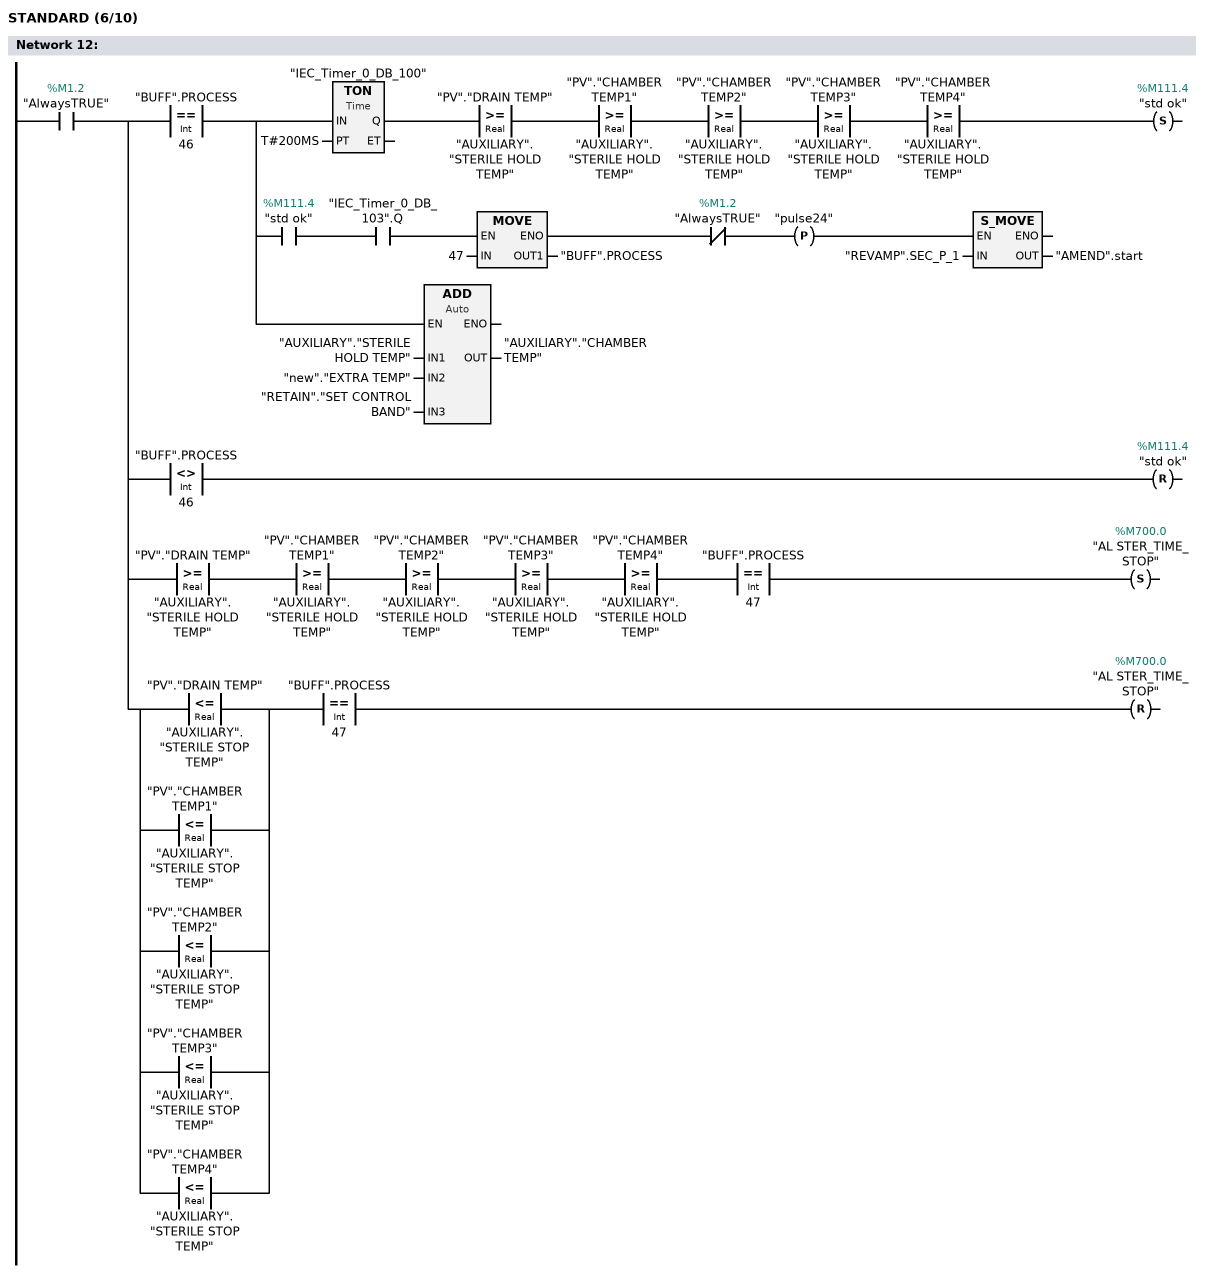
   RUNG wire#powerrail
      Contact( "AlwaysTRUE" )
      wire#w1
      { S7_Templates := "SrcType := Int" } EQ_Contact(in1 := "BUFF".PROCESS, in2 := 46)
      wire#w2
      { S7_Templates := "time_type := Time" } "IEC_Timer_0_DB_100".TON(pt := T#200MS, et =>)
      { S7_Templates := "SrcType := Real" } GE_Contact(in1 := "PV"."DRAIN TEMP", in2 := "AUXILIARY"."STERILE HOLD TEMP")
      { S7_Templates := "SrcType := Real" } GE_Contact(in1 := "PV"."CHAMBER TEMP1", in2 := "AUXILIARY"."STERILE HOLD TEMP")
      { S7_Templates := "SrcType := Real" } GE_Contact(in1 := "PV"."CHAMBER TEMP2", in2 := "AUXILIARY"."STERILE HOLD TEMP")
      { S7_Templates := "SrcType := Real" } GE_Contact(in1 := "PV"."CHAMBER TEMP3", in2 := "AUXILIARY"."STERILE HOLD TEMP")
      { S7_Templates := "SrcType := Real" } GE_Contact(in1 := "PV"."CHAMBER TEMP4", in2 := "AUXILIARY"."STERILE HOLD TEMP")
      S_Coil( "std ok" )
   END_RUNG
   RUNG wire#w2
      Contact( "std ok" )
      Contact( "IEC_Timer_0_DB_103".Q )
      Move(in := 47, out1 => "BUFF".PROCESS)
      I_Contact( "AlwaysTRUE" )
      P_Trig( "pulse24" )
      S_Move(in := "REVAMP".SEC_P_1, out => "AMEND".start)
   END_RUNG
   RUNG wire#w2
      Add(in1 := "AUXILIARY"."STERILE HOLD TEMP", in2 := "new"."EXTRA TEMP", in3 := "RETAIN"."SET CONTROL BAND", out => "AUXILIARY"."CHAMBER TEMP")
   END_RUNG
   RUNG wire#w1
      { S7_Templates := "SrcType := Int" } NE_Contact(in1 := "BUFF".PROCESS, in2 := 46)
      R_Coil( "std ok" )
   END_RUNG
   RUNG wire#w1
      { S7_Templates := "SrcType := Real" } GE_Contact(in1 := "PV"."DRAIN TEMP", in2 := "AUXILIARY"."STERILE HOLD TEMP")
      { S7_Templates := "SrcType := Real" } GE_Contact(in1 := "PV"."CHAMBER TEMP1", in2 := "AUXILIARY"."STERILE HOLD TEMP")
      { S7_Templates := "SrcType := Real" } GE_Contact(in1 := "PV"."CHAMBER TEMP2", in2 := "AUXILIARY"."STERILE HOLD TEMP")
      { S7_Templates := "SrcType := Real" } GE_Contact(in1 := "PV"."CHAMBER TEMP3", in2 := "AUXILIARY"."STERILE HOLD TEMP")
      { S7_Templates := "SrcType := Real" } GE_Contact(in1 := "PV"."CHAMBER TEMP4", in2 := "AUXILIARY"."STERILE HOLD TEMP")
      { S7_Templates := "SrcType := Int" } EQ_Contact(in1 := "BUFF".PROCESS, in2 := 47)
      S_Coil( "AL STER_TIME_STOP" )
   END_RUNG
   RUNG wire#w1
      { S7_Templates := "SrcType := Real" } LE_Contact(in1 := "PV"."DRAIN TEMP", in2 := "AUXILIARY"."STERILE STOP TEMP")
      wire#w3
      { S7_Templates := "SrcType := Int" } EQ_Contact(in1 := "BUFF".PROCESS, in2 := 47)
      R_Coil( "AL STER_TIME_STOP" )
   END_RUNG
   RUNG wire#w1
      { S7_Templates := "SrcType := Real" } LE_Contact(in1 := "PV"."CHAMBER TEMP1", in2 := "AUXILIARY"."STERILE STOP TEMP")
   END_RUNG wire#w3
   RUNG wire#w1
      { S7_Templates := "SrcType := Real" } LE_Contact(in1 := "PV"."CHAMBER TEMP2", in2 := "AUXILIARY"."STERILE STOP TEMP")
   END_RUNG wire#w3
   RUNG wire#w1
      { S7_Templates := "SrcType := Real" } LE_Contact(in1 := "PV"."CHAMBER TEMP3", in2 := "AUXILIARY"."STERILE STOP TEMP")
   END_RUNG wire#w3
   RUNG wire#w1
      { S7_Templates := "SrcType := Real" } LE_Contact(in1 := "PV"."CHAMBER TEMP4", in2 := "AUXILIARY"."STERILE STOP TEMP")
   END_RUNG wire#w3
   // the same network as SCL:
   #_w1 := "AlwaysTRUE" AND ("BUFF".PROCESS = 46);
   "IEC_Timer_0_DB_100".TON(IN := #_w1, PT := T#200MS);
   IF "IEC_Timer_0_DB_100".Q AND ("PV"."DRAIN TEMP" >= "AUXILIARY"."STERILE HOLD TEMP") AND ("PV"."CHAMBER TEMP1" >= "AUXILIARY"."STERILE HOLD TEMP") AND ("PV"."CHAMBER TEMP2" >= "AUXILIARY"."STERILE HOLD TEMP") AND ("PV"."CHAMBER TEMP3" >= "AUXILIARY"."STERILE HOLD TEMP") AND ("PV"."CHAMBER TEMP4" >= "AUXILIARY"."STERILE HOLD TEMP") THEN
       "std ok" := TRUE;
   END_IF;
   #_w2 := #_w1 AND "std ok" AND "IEC_Timer_0_DB_103".Q;
   IF #_w2 THEN "BUFF".PROCESS := 47; END_IF;
   #_w3 := #_w2 AND NOT "AlwaysTRUE";
   #_w4 := #_w3 AND NOT "pulse24";   // rising edge
   "pulse24" := #_w3;
   IF #_w4 THEN "AMEND".start := "REVAMP".SEC_P_1; END_IF;
   IF #_w1 THEN
       "AUXILIARY"."CHAMBER TEMP" := "AUXILIARY"."STERILE HOLD TEMP" + "new"."EXTRA TEMP" + "RETAIN"."SET CONTROL BAND";
   END_IF;
   IF "AlwaysTRUE" AND ("BUFF".PROCESS <> 46) THEN "std ok" := FALSE; END_IF;
   IF "AlwaysTRUE" AND ("PV"."DRAIN TEMP" >= "AUXILIARY"."STERILE HOLD TEMP") AND ("PV"."CHAMBER TEMP1" >= "AUXILIARY"."STERILE HOLD TEMP") AND ("PV"."CHAMBER TEMP2" >= "AUXILIARY"."STERILE HOLD TEMP") AND ("PV"."CHAMBER TEMP3" >= "AUXILIARY"."STERILE HOLD TEMP") AND ("PV"."CHAMBER TEMP4" >= "AUXILIARY"."STERILE HOLD TEMP") AND ("BUFF".PROCESS = 47) THEN
       "AL STER_TIME_STOP" := TRUE;
   END_IF;
   IF "AlwaysTRUE" AND (("PV"."DRAIN TEMP" <= "AUXILIARY"."STERILE STOP TEMP") OR ("PV"."CHAMBER TEMP1" <= "AUXILIARY"."STERILE STOP TEMP") OR ("PV"."CHAMBER TEMP2" <= "AUXILIARY"."STERILE STOP TEMP") OR ("PV"."CHAMBER TEMP3" <= "AUXILIARY"."STERILE STOP TEMP") OR ("PV"."CHAMBER TEMP4" <= "AUXILIARY"."STERILE STOP TEMP")) AND ("BUFF".PROCESS = 47) THEN
       "AL STER_TIME_STOP" := FALSE;
   END_IF;
END_REGION

REGION Network 13
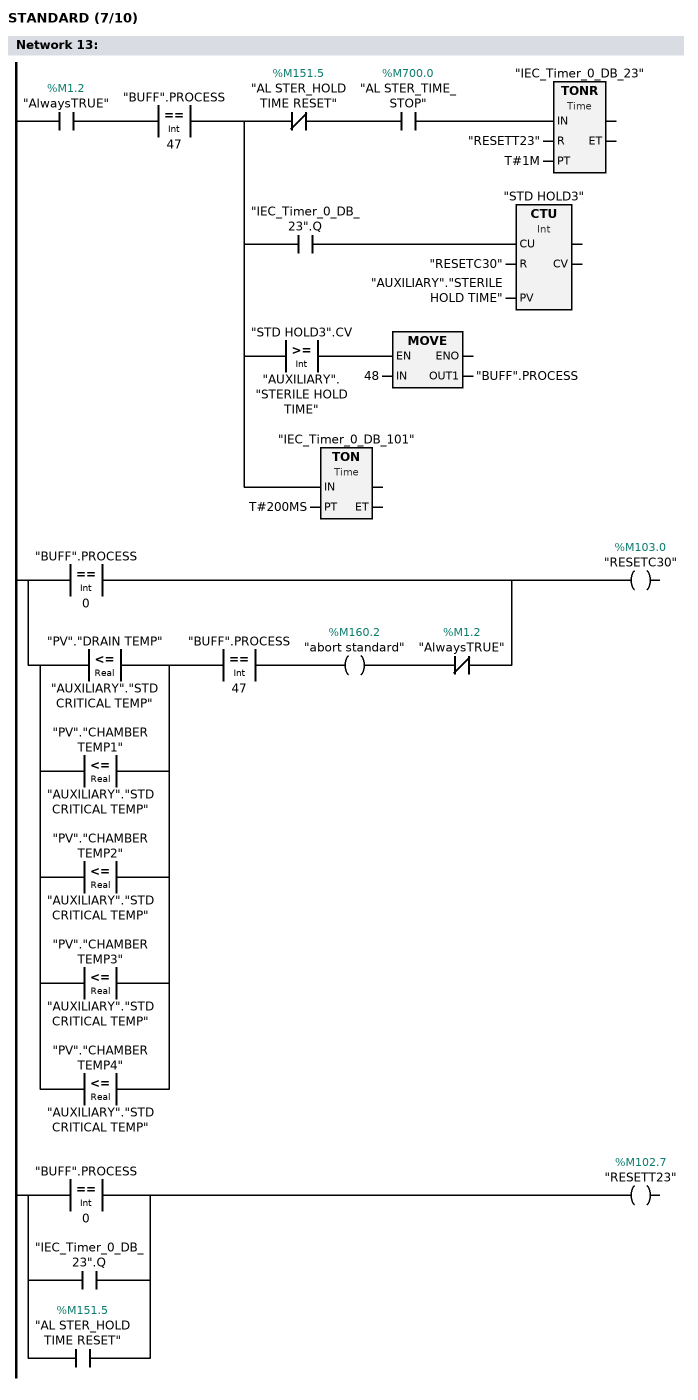
   RUNG wire#powerrail
      Contact( "AlwaysTRUE" )
      { S7_Templates := "SrcType := Int" } EQ_Contact(in1 := "BUFF".PROCESS, in2 := 47)
      wire#w1
      I_Contact( "AL STER_HOLD TIME RESET" )
      Contact( "AL STER_TIME_STOP" )
      { S7_Templates := "time_type := Time" } "IEC_Timer_0_DB_23".TONR(r := "RESETT23", pt := T#1M, et =>)
   END_RUNG
   RUNG wire#w1
      Contact( "IEC_Timer_0_DB_23".Q )
      { S7_Templates := "value_type := Int" } "STD HOLD3".CTU(r := "RESETC30", pv := "AUXILIARY"."STERILE HOLD TIME", cv =>)
   END_RUNG
   RUNG wire#w1
      { S7_Templates := "SrcType := Int" } GE_Contact(in1 := "STD HOLD3".CV, in2 := "AUXILIARY"."STERILE HOLD TIME")
      Move(in := 48, out1 => "BUFF".PROCESS)
   END_RUNG
   RUNG wire#w1
      { S7_Templates := "time_type := Time" } "IEC_Timer_0_DB_101".TON(pt := T#200MS, et =>)
   END_RUNG
   RUNG wire#powerrail
      { S7_Templates := "SrcType := Int" } EQ_Contact(in1 := "BUFF".PROCESS, in2 := 0)
      wire#w2
      Coil( "RESETC30" )
   END_RUNG
   RUNG wire#powerrail
      { S7_Templates := "SrcType := Real" } LE_Contact(in1 := "PV"."DRAIN TEMP", in2 := "AUXILIARY"."STD CRITICAL TEMP")
      wire#w3
      { S7_Templates := "SrcType := Int" } EQ_Contact(in1 := "BUFF".PROCESS, in2 := 47)
      Coil( "abort standard" )
      I_Contact( "AlwaysTRUE" )
   END_RUNG wire#w2
   RUNG wire#powerrail
      { S7_Templates := "SrcType := Real" } LE_Contact(in1 := "PV"."CHAMBER TEMP1", in2 := "AUXILIARY"."STD CRITICAL TEMP")
   END_RUNG wire#w3
   RUNG wire#powerrail
      { S7_Templates := "SrcType := Real" } LE_Contact(in1 := "PV"."CHAMBER TEMP2", in2 := "AUXILIARY"."STD CRITICAL TEMP")
   END_RUNG wire#w3
   RUNG wire#powerrail
      { S7_Templates := "SrcType := Real" } LE_Contact(in1 := "PV"."CHAMBER TEMP3", in2 := "AUXILIARY"."STD CRITICAL TEMP")
   END_RUNG wire#w3
   RUNG wire#powerrail
      { S7_Templates := "SrcType := Real" } LE_Contact(in1 := "PV"."CHAMBER TEMP4", in2 := "AUXILIARY"."STD CRITICAL TEMP")
   END_RUNG wire#w3
   RUNG wire#powerrail
      { S7_Templates := "SrcType := Int" } EQ_Contact(in1 := "BUFF".PROCESS, in2 := 0)
      wire#w4
      Coil( "RESETT23" )
   END_RUNG
   RUNG wire#powerrail
      Contact( "IEC_Timer_0_DB_23".Q )
   END_RUNG wire#w4
   RUNG wire#powerrail
      Contact( "AL STER_HOLD TIME RESET" )
   END_RUNG wire#w4
   // the same network as SCL:
   #_w1 := "AlwaysTRUE" AND ("BUFF".PROCESS = 47);
   "IEC_Timer_0_DB_23".TONR(IN := #_w1 AND NOT "AL STER_HOLD TIME RESET" AND "AL STER_TIME_STOP",
                           R := "RESETT23",
                           PT := T#1M);
   "STD HOLD3".CTU(CU := #_w1 AND "IEC_Timer_0_DB_23".Q, R := "RESETC30", PV := "AUXILIARY"."STERILE HOLD TIME");
   IF #_w1 AND ("STD HOLD3".CV >= "AUXILIARY"."STERILE HOLD TIME") THEN "BUFF".PROCESS := 48; END_IF;
   "IEC_Timer_0_DB_101".TON(IN := #_w1, PT := T#200MS);
   "abort standard" := (("PV"."DRAIN TEMP" <= "AUXILIARY"."STD CRITICAL TEMP") OR ("PV"."CHAMBER TEMP1" <= "AUXILIARY"."STD CRITICAL TEMP") OR ("PV"."CHAMBER TEMP2" <= "AUXILIARY"."STD CRITICAL TEMP") OR ("PV"."CHAMBER TEMP3" <= "AUXILIARY"."STD CRITICAL TEMP") OR ("PV"."CHAMBER TEMP4" <= "AUXILIARY"."STD CRITICAL TEMP")) AND ("BUFF".PROCESS = 47);
   "RESETC30" := ("BUFF".PROCESS = 0) OR ("abort standard" AND NOT "AlwaysTRUE");
   "RESETT23" := ("BUFF".PROCESS = 0) OR "IEC_Timer_0_DB_23".Q OR "AL STER_HOLD TIME RESET";
END_REGION

REGION Network 14
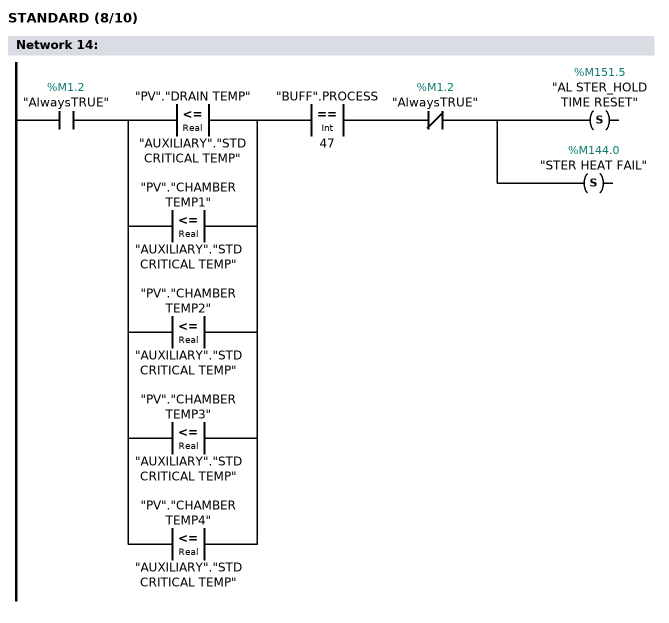
   RUNG wire#powerrail
      Contact( "AlwaysTRUE" )
      wire#w1
      { S7_Templates := "SrcType := Real" } LE_Contact(in1 := "PV"."DRAIN TEMP", in2 := "AUXILIARY"."STD CRITICAL TEMP")
      wire#w2
      { S7_Templates := "SrcType := Int" } EQ_Contact(in1 := "BUFF".PROCESS, in2 := 47)
      I_Contact( "AlwaysTRUE" )
      wire#w3
      S_Coil( "AL STER_HOLD TIME RESET" )
   END_RUNG
   RUNG wire#w1
      { S7_Templates := "SrcType := Real" } LE_Contact(in1 := "PV"."CHAMBER TEMP1", in2 := "AUXILIARY"."STD CRITICAL TEMP")
   END_RUNG wire#w2
   RUNG wire#w1
      { S7_Templates := "SrcType := Real" } LE_Contact(in1 := "PV"."CHAMBER TEMP2", in2 := "AUXILIARY"."STD CRITICAL TEMP")
   END_RUNG wire#w2
   RUNG wire#w1
      { S7_Templates := "SrcType := Real" } LE_Contact(in1 := "PV"."CHAMBER TEMP3", in2 := "AUXILIARY"."STD CRITICAL TEMP")
   END_RUNG wire#w2
   RUNG wire#w1
      { S7_Templates := "SrcType := Real" } LE_Contact(in1 := "PV"."CHAMBER TEMP4", in2 := "AUXILIARY"."STD CRITICAL TEMP")
   END_RUNG wire#w2
   RUNG wire#w3
      S_Coil( "STER HEAT FAIL" )
   END_RUNG
   // the same network as SCL:
   IF "AlwaysTRUE" AND (("PV"."DRAIN TEMP" <= "AUXILIARY"."STD CRITICAL TEMP") OR ("PV"."CHAMBER TEMP1" <= "AUXILIARY"."STD CRITICAL TEMP") OR ("PV"."CHAMBER TEMP2" <= "AUXILIARY"."STD CRITICAL TEMP") OR ("PV"."CHAMBER TEMP3" <= "AUXILIARY"."STD CRITICAL TEMP") OR ("PV"."CHAMBER TEMP4" <= "AUXILIARY"."STD CRITICAL TEMP")) AND ("BUFF".PROCESS = 47) AND NOT "AlwaysTRUE" THEN
       "AL STER_HOLD TIME RESET" := TRUE;
       "STER HEAT FAIL" := TRUE;
   END_IF;
END_REGION

REGION Network 15
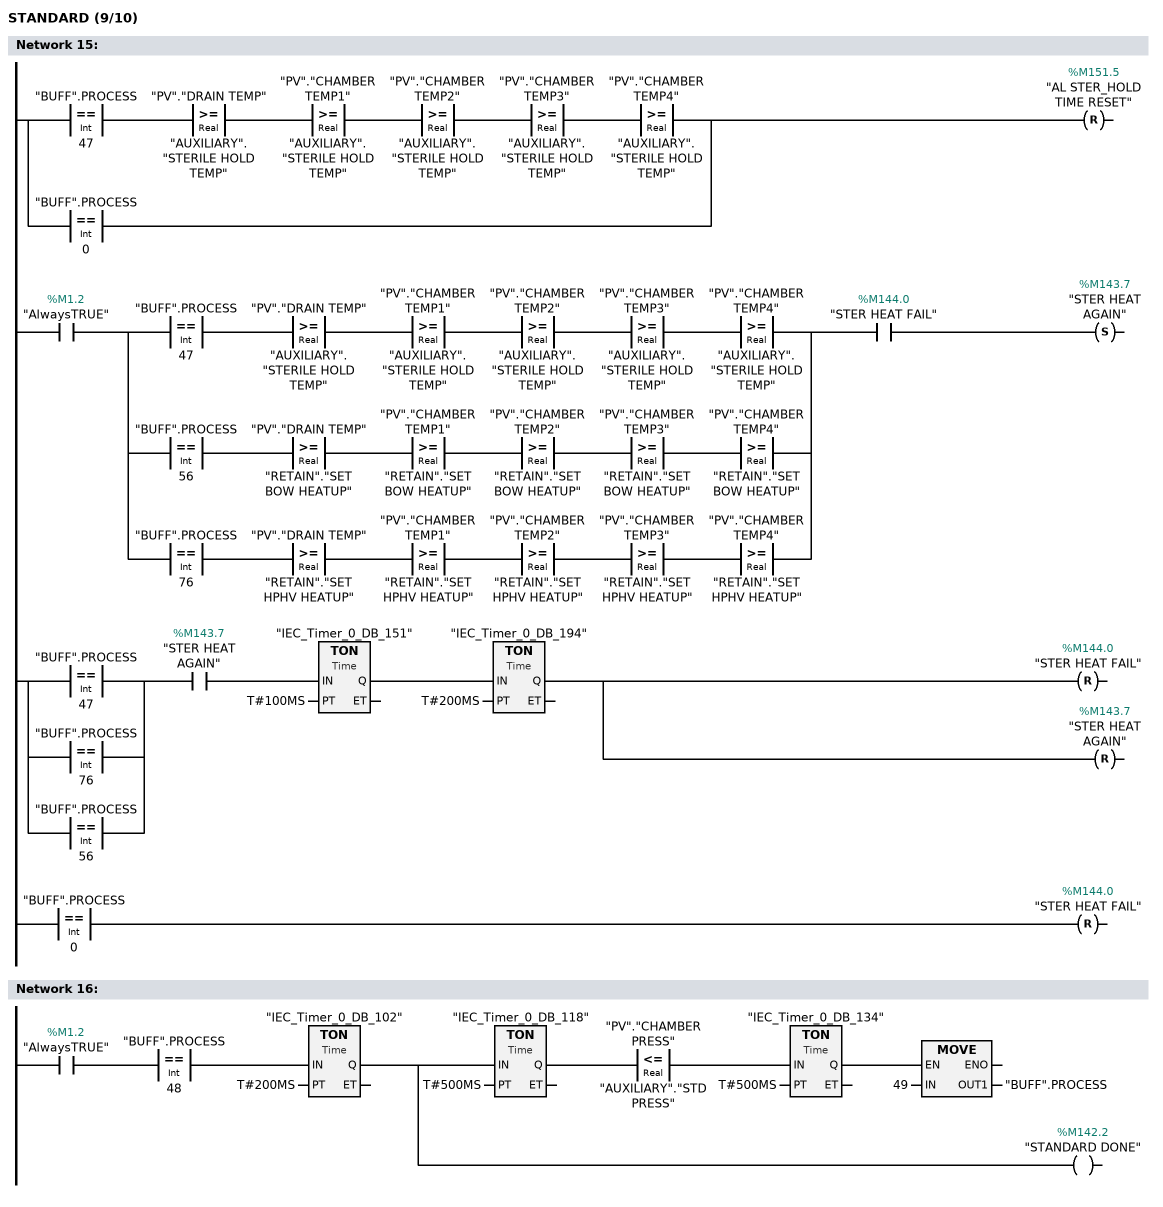
   RUNG wire#powerrail
      { S7_Templates := "SrcType := Int" } EQ_Contact(in1 := "BUFF".PROCESS, in2 := 47)
      { S7_Templates := "SrcType := Real" } GE_Contact(in1 := "PV"."DRAIN TEMP", in2 := "AUXILIARY"."STERILE HOLD TEMP")
      { S7_Templates := "SrcType := Real" } GE_Contact(in1 := "PV"."CHAMBER TEMP1", in2 := "AUXILIARY"."STERILE HOLD TEMP")
      { S7_Templates := "SrcType := Real" } GE_Contact(in1 := "PV"."CHAMBER TEMP2", in2 := "AUXILIARY"."STERILE HOLD TEMP")
      { S7_Templates := "SrcType := Real" } GE_Contact(in1 := "PV"."CHAMBER TEMP3", in2 := "AUXILIARY"."STERILE HOLD TEMP")
      { S7_Templates := "SrcType := Real" } GE_Contact(in1 := "PV"."CHAMBER TEMP4", in2 := "AUXILIARY"."STERILE HOLD TEMP")
      wire#w1
      R_Coil( "AL STER_HOLD TIME RESET" )
   END_RUNG
   RUNG wire#powerrail
      { S7_Templates := "SrcType := Int" } EQ_Contact(in1 := "BUFF".PROCESS, in2 := 0)
   END_RUNG wire#w1
   RUNG wire#powerrail
      Contact( "AlwaysTRUE" )
      wire#w2
      { S7_Templates := "SrcType := Int" } EQ_Contact(in1 := "BUFF".PROCESS, in2 := 47)
      { S7_Templates := "SrcType := Real" } GE_Contact(in1 := "PV"."DRAIN TEMP", in2 := "AUXILIARY"."STERILE HOLD TEMP")
      { S7_Templates := "SrcType := Real" } GE_Contact(in1 := "PV"."CHAMBER TEMP1", in2 := "AUXILIARY"."STERILE HOLD TEMP")
      { S7_Templates := "SrcType := Real" } GE_Contact(in1 := "PV"."CHAMBER TEMP2", in2 := "AUXILIARY"."STERILE HOLD TEMP")
      { S7_Templates := "SrcType := Real" } GE_Contact(in1 := "PV"."CHAMBER TEMP3", in2 := "AUXILIARY"."STERILE HOLD TEMP")
      { S7_Templates := "SrcType := Real" } GE_Contact(in1 := "PV"."CHAMBER TEMP4", in2 := "AUXILIARY"."STERILE HOLD TEMP")
      wire#w3
      Contact( "STER HEAT FAIL" )
      S_Coil( "STER HEAT AGAIN" )
   END_RUNG
   RUNG wire#w2
      { S7_Templates := "SrcType := Int" } EQ_Contact(in1 := "BUFF".PROCESS, in2 := 56)
      { S7_Templates := "SrcType := Real" } GE_Contact(in1 := "PV"."DRAIN TEMP", in2 := "RETAIN"."SET BOW HEATUP")
      { S7_Templates := "SrcType := Real" } GE_Contact(in1 := "PV"."CHAMBER TEMP1", in2 := "RETAIN"."SET BOW HEATUP")
      { S7_Templates := "SrcType := Real" } GE_Contact(in1 := "PV"."CHAMBER TEMP2", in2 := "RETAIN"."SET BOW HEATUP")
      { S7_Templates := "SrcType := Real" } GE_Contact(in1 := "PV"."CHAMBER TEMP3", in2 := "RETAIN"."SET BOW HEATUP")
      { S7_Templates := "SrcType := Real" } GE_Contact(in1 := "PV"."CHAMBER TEMP4", in2 := "RETAIN"."SET BOW HEATUP")
   END_RUNG wire#w3
   RUNG wire#w2
      { S7_Templates := "SrcType := Int" } EQ_Contact(in1 := "BUFF".PROCESS, in2 := 76)
      { S7_Templates := "SrcType := Real" } GE_Contact(in1 := "PV"."DRAIN TEMP", in2 := "RETAIN"."SET HPHV HEATUP")
      { S7_Templates := "SrcType := Real" } GE_Contact(in1 := "PV"."CHAMBER TEMP1", in2 := "RETAIN"."SET HPHV HEATUP")
      { S7_Templates := "SrcType := Real" } GE_Contact(in1 := "PV"."CHAMBER TEMP2", in2 := "RETAIN"."SET HPHV HEATUP")
      { S7_Templates := "SrcType := Real" } GE_Contact(in1 := "PV"."CHAMBER TEMP3", in2 := "RETAIN"."SET HPHV HEATUP")
      { S7_Templates := "SrcType := Real" } GE_Contact(in1 := "PV"."CHAMBER TEMP4", in2 := "RETAIN"."SET HPHV HEATUP")
   END_RUNG wire#w3
   RUNG wire#powerrail
      { S7_Templates := "SrcType := Int" } EQ_Contact(in1 := "BUFF".PROCESS, in2 := 47)
      wire#w4
      Contact( "STER HEAT AGAIN" )
      { S7_Templates := "time_type := Time" } "IEC_Timer_0_DB_151".TON(pt := T#100MS, et =>)
      { S7_Templates := "time_type := Time" } "IEC_Timer_0_DB_194".TON(pt := T#200MS, et =>)
      wire#w5
      R_Coil( "STER HEAT FAIL" )
   END_RUNG
   RUNG wire#powerrail
      { S7_Templates := "SrcType := Int" } EQ_Contact(in1 := "BUFF".PROCESS, in2 := 76)
   END_RUNG wire#w4
   RUNG wire#powerrail
      { S7_Templates := "SrcType := Int" } EQ_Contact(in1 := "BUFF".PROCESS, in2 := 56)
   END_RUNG wire#w4
   RUNG wire#w5
      R_Coil( "STER HEAT AGAIN" )
   END_RUNG
   RUNG wire#powerrail
      { S7_Templates := "SrcType := Int" } EQ_Contact(in1 := "BUFF".PROCESS, in2 := 0)
      R_Coil( "STER HEAT FAIL" )
   END_RUNG
   // the same network as SCL:
   IF (("BUFF".PROCESS = 47) AND ("PV"."DRAIN TEMP" >= "AUXILIARY"."STERILE HOLD TEMP") AND ("PV"."CHAMBER TEMP1" >= "AUXILIARY"."STERILE HOLD TEMP") AND ("PV"."CHAMBER TEMP2" >= "AUXILIARY"."STERILE HOLD TEMP") AND ("PV"."CHAMBER TEMP3" >= "AUXILIARY"."STERILE HOLD TEMP") AND ("PV"."CHAMBER TEMP4" >= "AUXILIARY"."STERILE HOLD TEMP")) OR ("BUFF".PROCESS = 0) THEN
       "AL STER_HOLD TIME RESET" := FALSE;
   END_IF;
   IF "AlwaysTRUE" AND ((("BUFF".PROCESS = 47) AND ("PV"."DRAIN TEMP" >= "AUXILIARY"."STERILE HOLD TEMP") AND ("PV"."CHAMBER TEMP1" >= "AUXILIARY"."STERILE HOLD TEMP") AND ("PV"."CHAMBER TEMP2" >= "AUXILIARY"."STERILE HOLD TEMP") AND ("PV"."CHAMBER TEMP3" >= "AUXILIARY"."STERILE HOLD TEMP") AND ("PV"."CHAMBER TEMP4" >= "AUXILIARY"."STERILE HOLD TEMP")) OR (("BUFF".PROCESS = 56) AND ("PV"."DRAIN TEMP" >= "RETAIN"."SET BOW HEATUP") AND ("PV"."CHAMBER TEMP1" >= "RETAIN"."SET BOW HEATUP") AND ("PV"."CHAMBER TEMP2" >= "RETAIN"."SET BOW HEATUP") AND ("PV"."CHAMBER TEMP3" >= "RETAIN"."SET BOW HEATUP") AND ("PV"."CHAMBER TEMP4" >= "RETAIN"."SET BOW HEATUP")) OR (("BUFF".PROCESS = 76) AND ("PV"."DRAIN TEMP" >= "RETAIN"."SET HPHV HEATUP") AND ("PV"."CHAMBER TEMP1" >= "RETAIN"."SET HPHV HEATUP") AND ("PV"."CHAMBER TEMP2" >= "RETAIN"."SET HPHV HEATUP") AND ("PV"."CHAMBER TEMP3" >= "RETAIN"."SET HPHV HEATUP") AND ("PV"."CHAMBER TEMP4" >= "RETAIN"."SET HPHV HEATUP"))) AND "STER HEAT FAIL" THEN
       "STER HEAT AGAIN" := TRUE;
   END_IF;
   "IEC_Timer_0_DB_151".TON(IN := (("BUFF".PROCESS = 47) OR ("BUFF".PROCESS = 76) OR ("BUFF".PROCESS = 56)) AND "STER HEAT AGAIN",
                           PT := T#100MS);
   "IEC_Timer_0_DB_194".TON(IN := "IEC_Timer_0_DB_151".Q, PT := T#200MS);
   IF "IEC_Timer_0_DB_194".Q THEN
       "STER HEAT FAIL" := FALSE;
       "STER HEAT AGAIN" := FALSE;
   END_IF;
   IF "BUFF".PROCESS = 0 THEN "STER HEAT FAIL" := FALSE; END_IF;
END_REGION

REGION Network 16
   RUNG wire#powerrail
      Contact( "AlwaysTRUE" )
      { S7_Templates := "SrcType := Int" } EQ_Contact(in1 := "BUFF".PROCESS, in2 := 48)
      { S7_Templates := "time_type := Time" } "IEC_Timer_0_DB_102".TON(pt := T#200MS, et =>)
      wire#w1
      { S7_Templates := "time_type := Time" } "IEC_Timer_0_DB_118".TON(pt := T#500MS, et =>)
      { S7_Templates := "SrcType := Real" } LE_Contact(in1 := "PV"."CHAMBER PRESS", in2 := "AUXILIARY"."STD PRESS")
      { S7_Templates := "time_type := Time" } "IEC_Timer_0_DB_134".TON(pt := T#500MS, et =>)
      Move(in := 49, out1 => "BUFF".PROCESS)
   END_RUNG
   RUNG wire#w1
      Coil( "STANDARD DONE" )
   END_RUNG
   // the same network as SCL:
   "IEC_Timer_0_DB_102".TON(IN := "AlwaysTRUE" AND ("BUFF".PROCESS = 48), PT := T#200MS);
   "IEC_Timer_0_DB_118".TON(IN := "IEC_Timer_0_DB_102".Q, PT := T#500MS);
   "IEC_Timer_0_DB_134".TON(IN := "IEC_Timer_0_DB_118".Q AND ("PV"."CHAMBER PRESS" <= "AUXILIARY"."STD PRESS"),
                           PT := T#500MS);
   IF "IEC_Timer_0_DB_134".Q THEN "BUFF".PROCESS := 49; END_IF;
   "STANDARD DONE" := "IEC_Timer_0_DB_102".Q;
END_REGION

REGION Network 17
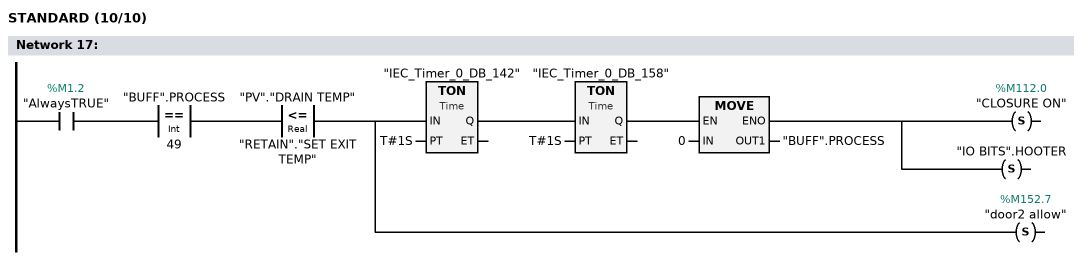
   RUNG wire#powerrail
      Contact( "AlwaysTRUE" )
      { S7_Templates := "SrcType := Int" } EQ_Contact(in1 := "BUFF".PROCESS, in2 := 49)
      { S7_Templates := "SrcType := Real" } LE_Contact(in1 := "PV"."DRAIN TEMP", in2 := "RETAIN"."SET EXIT TEMP")
      wire#w1
      { S7_Templates := "time_type := Time" } "IEC_Timer_0_DB_142".TON(pt := T#1S, et =>)
      { S7_Templates := "time_type := Time" } "IEC_Timer_0_DB_158".TON(pt := T#1S, et =>)
      Move(in := 0, out1 => "BUFF".PROCESS)
      wire#w2
      S_Coil( "CLOSURE ON" )
   END_RUNG
   RUNG wire#w2
      S_Coil( "IO BITS".HOOTER )
   END_RUNG
   RUNG wire#w1
      S_Coil( "door2 allow" )
   END_RUNG
   // the same network as SCL:
   #_w1 := "AlwaysTRUE" AND ("BUFF".PROCESS = 49) AND ("PV"."DRAIN TEMP" <= "RETAIN"."SET EXIT TEMP");
   "IEC_Timer_0_DB_142".TON(IN := #_w1, PT := T#1S);
   "IEC_Timer_0_DB_158".TON(IN := "IEC_Timer_0_DB_142".Q, PT := T#1S);
   IF "IEC_Timer_0_DB_158".Q THEN
       "BUFF".PROCESS := 0;
       "CLOSURE ON" := TRUE;
       "IO BITS".HOOTER := TRUE;
   END_IF;
   IF #_w1 THEN "door2 allow" := TRUE; END_IF;
END_REGION
END_FUNCTION

FUNCTION "VACCUM" : Void   // FC12, LAD
{ S7_Optimized_Access := 'TRUE' }
// stored: SetENOAutomatically false
   VAR_TEMP
      "VACCUM DIFF" : Real;
      "VACCUM LEAK DIFF" : Real;
   END_VAR
   VAR_TEMP   // added for the SCL form of the ladder/FBD networks
      _w1 : Bool;
      _w2 : Bool;
      _w3 : Bool;
      _w4 : Bool;
      _w5 : Bool;
      _w6 : Bool;
      _w7 : Bool;
      _w8 : Bool;
      _w9 : Bool;
      _w10 : Bool;
      _w11 : Bool;
      _w12 : Bool;
      _w13 : Bool;
      _w14 : Bool;
      _w15 : Bool;
      _w16 : Bool;
      _w17 : Bool;
      _w18 : Bool;
      _w19 : Bool;
      _w20 : Bool;
   END_VAR
BEGIN

REGION Network 1
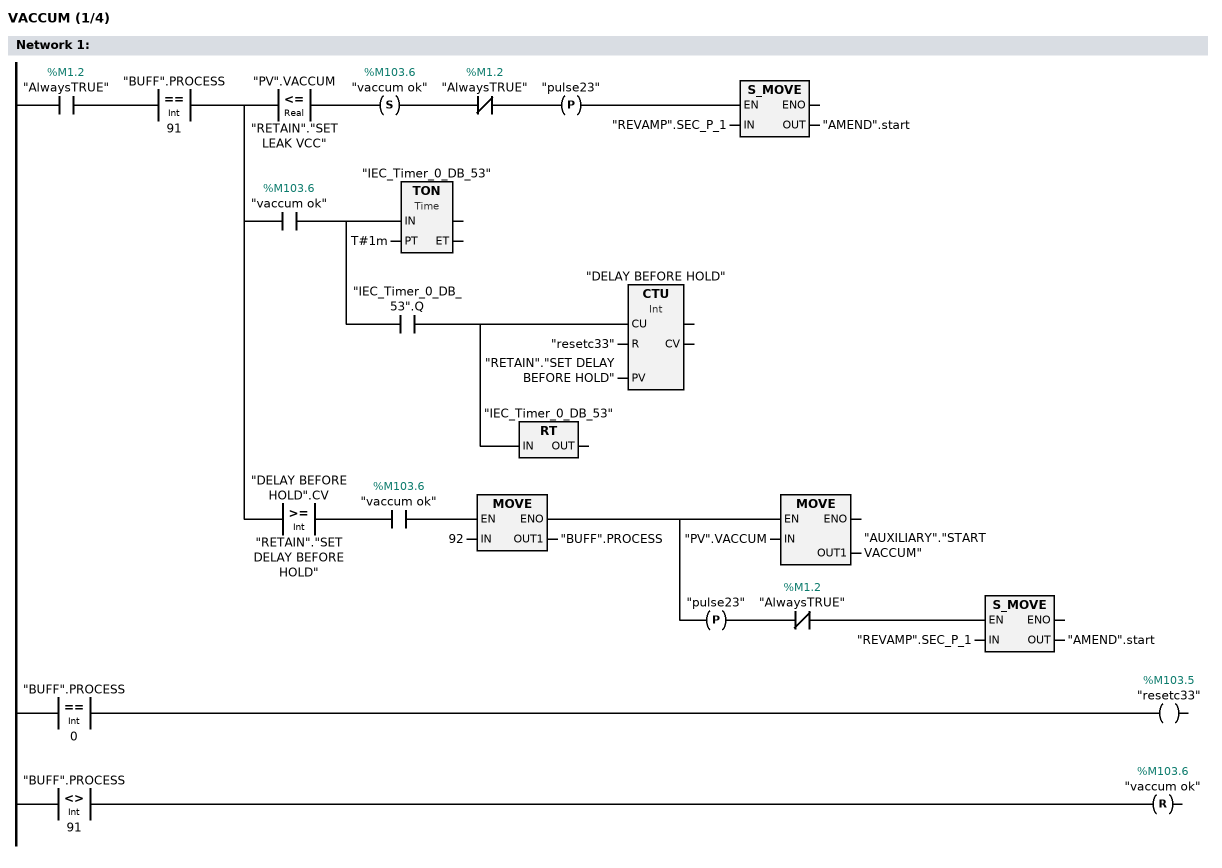
   RUNG wire#powerrail
      Contact( "AlwaysTRUE" )
      { S7_Templates := "SrcType := Int" } EQ_Contact(in1 := "BUFF".PROCESS, in2 := 91)
      wire#w1
      { S7_Templates := "SrcType := Real" } LE_Contact(in1 := "PV".VACCUM, in2 := "RETAIN"."SET LEAK VCC")
      S_Coil( "vaccum ok" )
      I_Contact( "AlwaysTRUE" )
      P_Trig( "pulse23" )
      S_Move(in := "REVAMP".SEC_P_1, out => "AMEND".start)
   END_RUNG
   RUNG wire#w1
      Contact( "vaccum ok" )
      wire#w2
      { S7_Templates := "time_type := Time" } "IEC_Timer_0_DB_53".TON(pt := T#1m, et =>)
   END_RUNG
   RUNG wire#w2
      Contact( "IEC_Timer_0_DB_53".Q )
      wire#w3
      { S7_Templates := "value_type := Int" } "DELAY BEFORE HOLD".CTU(r := "resetc33", pv := "RETAIN"."SET DELAY BEFORE HOLD", cv =>)
   END_RUNG
   RUNG wire#w3
      RT_Coil( "IEC_Timer_0_DB_53" )
   END_RUNG
   RUNG wire#w1
      { S7_Templates := "SrcType := Int" } GE_Contact(in1 := "DELAY BEFORE HOLD".CV, in2 := "RETAIN"."SET DELAY BEFORE HOLD")
      Contact( "vaccum ok" )
      Move(in := 92, out1 => "BUFF".PROCESS)
      wire#w4
      Move(in := "PV".VACCUM, out1 => "AUXILIARY"."START VACCUM")
   END_RUNG
   RUNG wire#w4
      P_Trig( "pulse23" )
      I_Contact( "AlwaysTRUE" )
      S_Move(in := "REVAMP".SEC_P_1, out => "AMEND".start)
   END_RUNG
   RUNG wire#powerrail
      { S7_Templates := "SrcType := Int" } EQ_Contact(in1 := "BUFF".PROCESS, in2 := 0)
      Coil( "resetc33" )
   END_RUNG
   RUNG wire#powerrail
      { S7_Templates := "SrcType := Int" } NE_Contact(in1 := "BUFF".PROCESS, in2 := 91)
      R_Coil( "vaccum ok" )
   END_RUNG
   // the same network as SCL:
   #_w1 := "AlwaysTRUE" AND ("BUFF".PROCESS = 91);
   #_w2 := #_w1 AND ("PV".VACCUM <= "RETAIN"."SET LEAK VCC");
   IF #_w2 THEN "vaccum ok" := TRUE; END_IF;
   #_w3 := #_w2 AND NOT "AlwaysTRUE";
   #_w4 := #_w3 AND NOT "pulse23";   // rising edge
   "pulse23" := #_w3;
   IF #_w4 THEN "AMEND".start := "REVAMP".SEC_P_1; END_IF;
   #_w5 := #_w1 AND "vaccum ok";
   "IEC_Timer_0_DB_53".TON(IN := #_w5, PT := T#1m);
   #_w6 := #_w5 AND "IEC_Timer_0_DB_53".Q;
   "DELAY BEFORE HOLD".CTU(CU := #_w6, R := "resetc33", PV := "RETAIN"."SET DELAY BEFORE HOLD");
   IF #_w6 THEN RESET_TIMER("IEC_Timer_0_DB_53"); END_IF;
   #_w7 := #_w1 AND ("DELAY BEFORE HOLD".CV >= "RETAIN"."SET DELAY BEFORE HOLD") AND "vaccum ok";
   IF #_w7 THEN
       "BUFF".PROCESS := 92;
       "AUXILIARY"."START VACCUM" := "PV".VACCUM;
   END_IF;
   #_w8 := #_w7 AND NOT "pulse23";   // rising edge
   "pulse23" := #_w7;
   IF #_w8 AND NOT "AlwaysTRUE" THEN "AMEND".start := "REVAMP".SEC_P_1; END_IF;
   "resetc33" := "BUFF".PROCESS = 0;
   IF "BUFF".PROCESS <> 91 THEN "vaccum ok" := FALSE; END_IF;
END_REGION

REGION Network 2
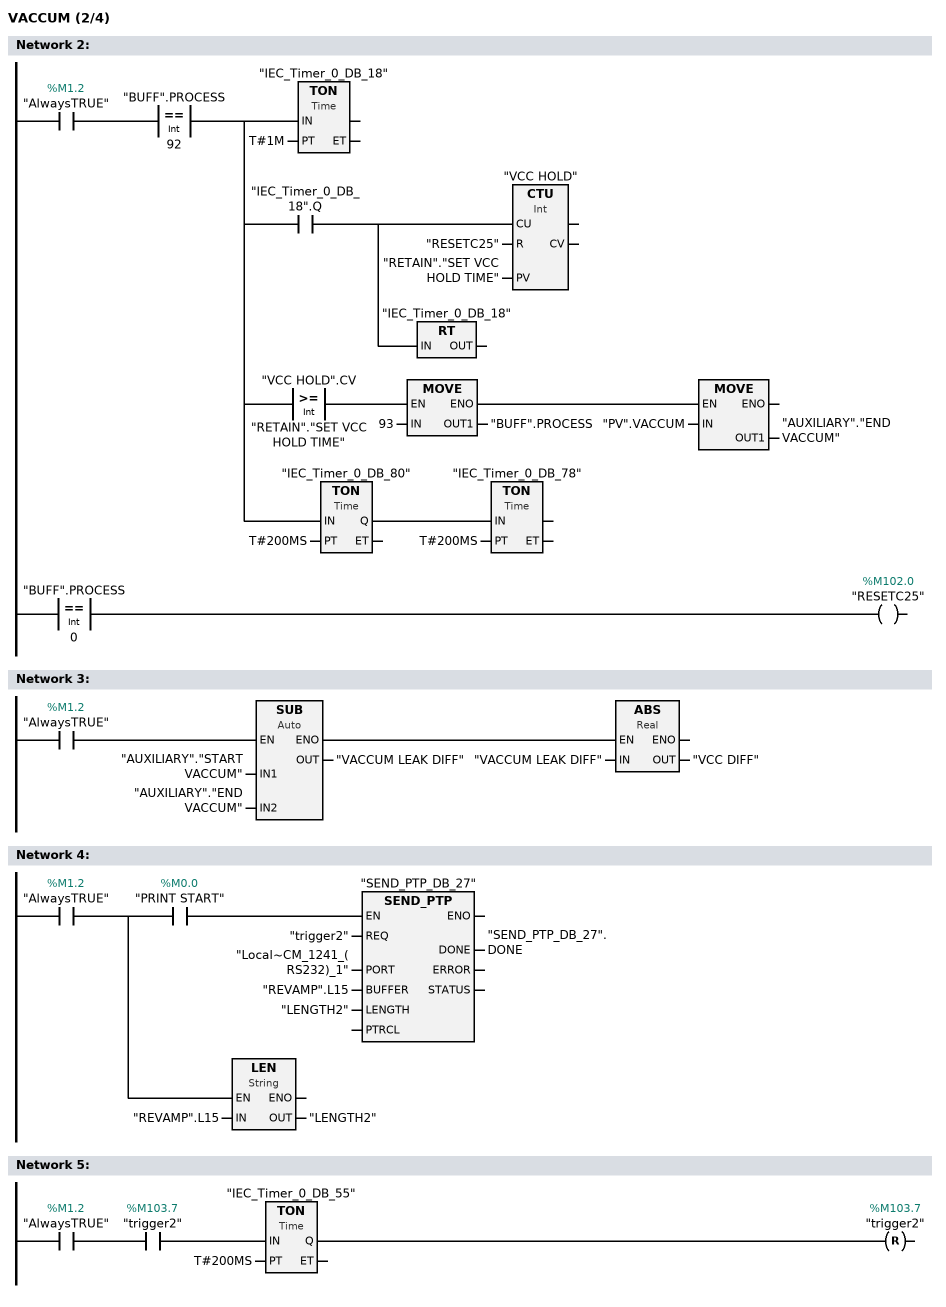
   RUNG wire#powerrail
      Contact( "AlwaysTRUE" )
      { S7_Templates := "SrcType := Int" } EQ_Contact(in1 := "BUFF".PROCESS, in2 := 92)
      wire#w1
      { S7_Templates := "time_type := Time" } "IEC_Timer_0_DB_18".TON(pt := T#1M, et =>)
   END_RUNG
   RUNG wire#w1
      Contact( "IEC_Timer_0_DB_18".Q )
      wire#w2
      { S7_Templates := "value_type := Int" } "VCC HOLD".CTU(r := "RESETC25", pv := "RETAIN"."SET VCC HOLD TIME", cv =>)
   END_RUNG
   RUNG wire#w2
      RT_Coil( "IEC_Timer_0_DB_18" )
   END_RUNG
   RUNG wire#w1
      { S7_Templates := "SrcType := Int" } GE_Contact(in1 := "VCC HOLD".CV, in2 := "RETAIN"."SET VCC HOLD TIME")
      Move(in := 93, out1 => "BUFF".PROCESS)
      Move(in := "PV".VACCUM, out1 => "AUXILIARY"."END VACCUM")
   END_RUNG
   RUNG wire#w1
      { S7_Templates := "time_type := Time" } "IEC_Timer_0_DB_80".TON(pt := T#200MS, et =>)
      { S7_Templates := "time_type := Time" } "IEC_Timer_0_DB_78".TON(pt := T#200MS, et =>)
   END_RUNG
   RUNG wire#powerrail
      { S7_Templates := "SrcType := Int" } EQ_Contact(in1 := "BUFF".PROCESS, in2 := 0)
      Coil( "RESETC25" )
   END_RUNG
   // the same network as SCL:
   #_w1 := "AlwaysTRUE" AND ("BUFF".PROCESS = 92);
   "IEC_Timer_0_DB_18".TON(IN := #_w1, PT := T#1M);
   #_w2 := #_w1 AND "IEC_Timer_0_DB_18".Q;
   "VCC HOLD".CTU(CU := #_w2, R := "RESETC25", PV := "RETAIN"."SET VCC HOLD TIME");
   IF #_w2 THEN RESET_TIMER("IEC_Timer_0_DB_18"); END_IF;
   IF #_w1 AND ("VCC HOLD".CV >= "RETAIN"."SET VCC HOLD TIME") THEN
       "BUFF".PROCESS := 93;
       "AUXILIARY"."END VACCUM" := "PV".VACCUM;
   END_IF;
   "IEC_Timer_0_DB_80".TON(IN := #_w1, PT := T#200MS);
   "IEC_Timer_0_DB_78".TON(IN := "IEC_Timer_0_DB_80".Q, PT := T#200MS);
   "RESETC25" := "BUFF".PROCESS = 0;
END_REGION

REGION Network 3
   RUNG wire#powerrail
      Contact( "AlwaysTRUE" )
      Sub(in1 := "AUXILIARY"."START VACCUM", in2 := "AUXILIARY"."END VACCUM", out => "VACCUM LEAK DIFF")
      { S7_Templates := "SrcType := Real" } Abs(in := "VACCUM LEAK DIFF", out => "VCC DIFF")
   END_RUNG
   // the same network as SCL:
   IF "AlwaysTRUE" THEN
       "VACCUM LEAK DIFF" := "AUXILIARY"."START VACCUM" - "AUXILIARY"."END VACCUM";
       "VCC DIFF" := ABS("VACCUM LEAK DIFF");
   END_IF;
END_REGION

REGION Network 4
   RUNG wire#powerrail
      Contact( "AlwaysTRUE" )
      wire#w1
      Contact( "PRINT START" )
      "SEND_PTP_DB_27".SEND_PTP(REQ := "trigger2", PORT := "Local~CM_1241_(RS232)_1", BUFFER := "REVAMP".L15, LENGTH := "LENGTH2", PTRCL :=, DONE => "SEND_PTP_DB_27".DONE, ERROR =>, STATUS =>)
   END_RUNG
   RUNG wire#w1
      { S7_Templates := "[str_type := String, return_type := Int]" } LEN(IN := "REVAMP".L15, OUT => "LENGTH2")
   END_RUNG
   // the same network as SCL:
   #_w1 := "AlwaysTRUE";
   IF "AlwaysTRUE" AND "PRINT START" THEN
       "SEND_PTP_DB_27"(REQ := "trigger2",   // SEND_PTP
                        PORT := "Local~CM_1241_(RS232)_1",
                        BUFFER := "REVAMP".L15,
                        LENGTH := "LENGTH2",
                        DONE => "SEND_PTP_DB_27".DONE);
   END_IF;
   IF #_w1 THEN LEN(IN := "REVAMP".L15, OUT => "LENGTH2"); END_IF;
END_REGION

REGION Network 5
   RUNG wire#powerrail
      Contact( "AlwaysTRUE" )
      Contact( "trigger2" )
      { S7_Templates := "time_type := Time" } "IEC_Timer_0_DB_55".TON(pt := T#200MS, et =>)
      R_Coil( "trigger2" )
   END_RUNG
   // the same network as SCL:
   "IEC_Timer_0_DB_55".TON(IN := "AlwaysTRUE" AND "trigger2", PT := T#200MS);
   IF "IEC_Timer_0_DB_55".Q THEN "trigger2" := FALSE; END_IF;
END_REGION

REGION Network 6
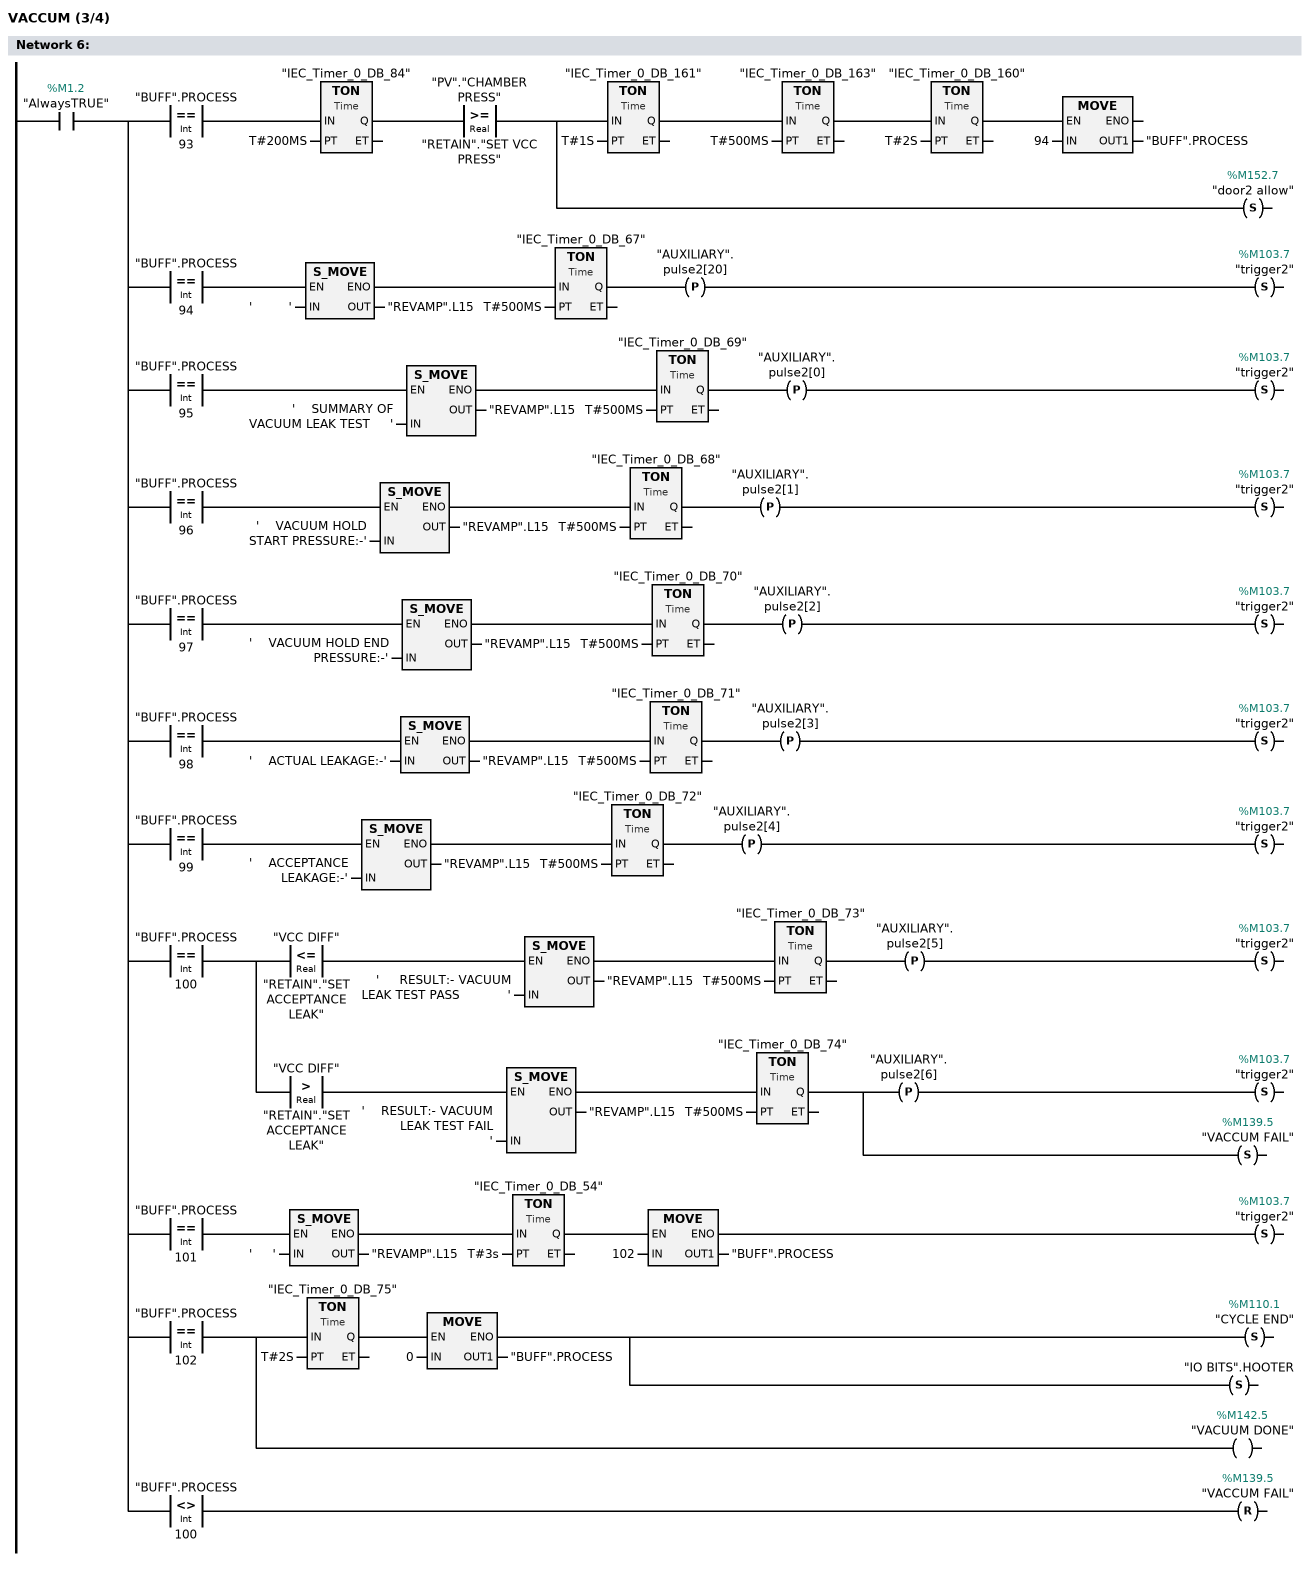
   RUNG wire#powerrail
      Contact( "AlwaysTRUE" )
      wire#w1
      { S7_Templates := "SrcType := Int" } EQ_Contact(in1 := "BUFF".PROCESS, in2 := 93)
      { S7_Templates := "time_type := Time" } "IEC_Timer_0_DB_84".TON(pt := T#200MS, et =>)
      { S7_Templates := "SrcType := Real" } GE_Contact(in1 := "PV"."CHAMBER PRESS", in2 := "RETAIN"."SET VCC PRESS")
      wire#w2
      { S7_Templates := "time_type := Time" } "IEC_Timer_0_DB_161".TON(pt := T#1S, et =>)
      { S7_Templates := "time_type := Time" } "IEC_Timer_0_DB_163".TON(pt := T#500MS, et =>)
      { S7_Templates := "time_type := Time" } "IEC_Timer_0_DB_160".TON(pt := T#2S, et =>)
      Move(in := 94, out1 => "BUFF".PROCESS)
   END_RUNG
   RUNG wire#w2
      S_Coil( "door2 allow" )
   END_RUNG
   RUNG wire#w1
      { S7_Templates := "SrcType := Int" } EQ_Contact(in1 := "BUFF".PROCESS, in2 := 94)
      S_Move(in := '         ', out => "REVAMP".L15)
      { S7_Templates := "time_type := Time" } "IEC_Timer_0_DB_67".TON(pt := T#500MS, et =>)
      P_Trig( "AUXILIARY".pulse2[20] )
      S_Coil( "trigger2" )
   END_RUNG
   RUNG wire#w1
      { S7_Templates := "SrcType := Int" } EQ_Contact(in1 := "BUFF".PROCESS, in2 := 95)
      S_Move(in := '    SUMMARY OF VACUUM LEAK TEST     ', out => "REVAMP".L15)
      { S7_Templates := "time_type := Time" } "IEC_Timer_0_DB_69".TON(pt := T#500MS, et =>)
      P_Trig( "AUXILIARY".pulse2[0] )
      S_Coil( "trigger2" )
   END_RUNG
   RUNG wire#w1
      { S7_Templates := "SrcType := Int" } EQ_Contact(in1 := "BUFF".PROCESS, in2 := 96)
      S_Move(in := '    VACUUM HOLD START PRESSURE:-', out => "REVAMP".L15)
      { S7_Templates := "time_type := Time" } "IEC_Timer_0_DB_68".TON(pt := T#500MS, et =>)
      P_Trig( "AUXILIARY".pulse2[1] )
      S_Coil( "trigger2" )
   END_RUNG
   RUNG wire#w1
      { S7_Templates := "SrcType := Int" } EQ_Contact(in1 := "BUFF".PROCESS, in2 := 97)
      S_Move(in := '    VACUUM HOLD END PRESSURE:-', out => "REVAMP".L15)
      { S7_Templates := "time_type := Time" } "IEC_Timer_0_DB_70".TON(pt := T#500MS, et =>)
      P_Trig( "AUXILIARY".pulse2[2] )
      S_Coil( "trigger2" )
   END_RUNG
   RUNG wire#w1
      { S7_Templates := "SrcType := Int" } EQ_Contact(in1 := "BUFF".PROCESS, in2 := 98)
      S_Move(in := '    ACTUAL LEAKAGE:-', out => "REVAMP".L15)
      { S7_Templates := "time_type := Time" } "IEC_Timer_0_DB_71".TON(pt := T#500MS, et =>)
      P_Trig( "AUXILIARY".pulse2[3] )
      S_Coil( "trigger2" )
   END_RUNG
   RUNG wire#w1
      { S7_Templates := "SrcType := Int" } EQ_Contact(in1 := "BUFF".PROCESS, in2 := 99)
      S_Move(in := '    ACCEPTANCE LEAKAGE:-', out => "REVAMP".L15)
      { S7_Templates := "time_type := Time" } "IEC_Timer_0_DB_72".TON(pt := T#500MS, et =>)
      P_Trig( "AUXILIARY".pulse2[4] )
      S_Coil( "trigger2" )
   END_RUNG
   RUNG wire#w1
      { S7_Templates := "SrcType := Int" } EQ_Contact(in1 := "BUFF".PROCESS, in2 := 100)
      wire#w3
      { S7_Templates := "SrcType := Real" } LE_Contact(in1 := "VCC DIFF", in2 := "RETAIN"."SET ACCEPTANCE LEAK")
      S_Move(in := '     RESULT:- VACUUM LEAK TEST PASS            ', out => "REVAMP".L15)
      { S7_Templates := "time_type := Time" } "IEC_Timer_0_DB_73".TON(pt := T#500MS, et =>)
      P_Trig( "AUXILIARY".pulse2[5] )
      S_Coil( "trigger2" )
   END_RUNG
   RUNG wire#w3
      { S7_Templates := "SrcType := Real" } GT_Contact(in1 := "VCC DIFF", in2 := "RETAIN"."SET ACCEPTANCE LEAK")
      S_Move(in := '    RESULT:- VACUUM LEAK TEST FAIL                   ', out => "REVAMP".L15)
      { S7_Templates := "time_type := Time" } "IEC_Timer_0_DB_74".TON(pt := T#500MS, et =>)
      wire#w4
      P_Trig( "AUXILIARY".pulse2[6] )
      S_Coil( "trigger2" )
   END_RUNG
   RUNG wire#w4
      S_Coil( "VACCUM FAIL" )
   END_RUNG
   RUNG wire#w1
      { S7_Templates := "SrcType := Int" } EQ_Contact(in1 := "BUFF".PROCESS, in2 := 101)
      S_Move(in := '     ', out => "REVAMP".L15)
      { S7_Templates := "time_type := Time" } "IEC_Timer_0_DB_54".TON(pt := T#3s, et =>)
      Move(in := 102, out1 => "BUFF".PROCESS)
      S_Coil( "trigger2" )
   END_RUNG
   RUNG wire#w1
      { S7_Templates := "SrcType := Int" } EQ_Contact(in1 := "BUFF".PROCESS, in2 := 102)
      wire#w5
      { S7_Templates := "time_type := Time" } "IEC_Timer_0_DB_75".TON(pt := T#2S, et =>)
      Move(in := 0, out1 => "BUFF".PROCESS)
      wire#w6
      S_Coil( "CYCLE END" )
   END_RUNG
   RUNG wire#w6
      S_Coil( "IO BITS".HOOTER )
   END_RUNG
   RUNG wire#w5
      Coil( "VACUUM DONE" )
   END_RUNG
   RUNG wire#w1
      { S7_Templates := "SrcType := Int" } NE_Contact(in1 := "BUFF".PROCESS, in2 := 100)
      R_Coil( "VACCUM FAIL" )
   END_RUNG
   // the same network as SCL:
   "IEC_Timer_0_DB_84".TON(IN := "AlwaysTRUE" AND ("BUFF".PROCESS = 93), PT := T#200MS);
   #_w1 := "IEC_Timer_0_DB_84".Q AND ("PV"."CHAMBER PRESS" >= "RETAIN"."SET VCC PRESS");
   "IEC_Timer_0_DB_161".TON(IN := #_w1, PT := T#1S);
   "IEC_Timer_0_DB_163".TON(IN := "IEC_Timer_0_DB_161".Q, PT := T#500MS);
   "IEC_Timer_0_DB_160".TON(IN := "IEC_Timer_0_DB_163".Q, PT := T#2S);
   IF "IEC_Timer_0_DB_160".Q THEN "BUFF".PROCESS := 94; END_IF;
   IF #_w1 THEN "door2 allow" := TRUE; END_IF;
   #_w2 := "AlwaysTRUE" AND ("BUFF".PROCESS = 94);
   IF #_w2 THEN "REVAMP".L15 := '         '; END_IF;
   "IEC_Timer_0_DB_67".TON(IN := #_w2, PT := T#500MS);
   #_w3 := "IEC_Timer_0_DB_67".Q AND NOT "AUXILIARY".pulse2[20];   // rising edge
   "AUXILIARY".pulse2[20] := "IEC_Timer_0_DB_67".Q;
   IF #_w3 THEN "trigger2" := TRUE; END_IF;
   #_w4 := "AlwaysTRUE" AND ("BUFF".PROCESS = 95);
   IF #_w4 THEN "REVAMP".L15 := '    SUMMARY OF VACUUM LEAK TEST     '; END_IF;
   "IEC_Timer_0_DB_69".TON(IN := #_w4, PT := T#500MS);
   #_w5 := "IEC_Timer_0_DB_69".Q AND NOT "AUXILIARY".pulse2[0];   // rising edge
   "AUXILIARY".pulse2[0] := "IEC_Timer_0_DB_69".Q;
   IF #_w5 THEN "trigger2" := TRUE; END_IF;
   #_w6 := "AlwaysTRUE" AND ("BUFF".PROCESS = 96);
   IF #_w6 THEN "REVAMP".L15 := '    VACUUM HOLD START PRESSURE:-'; END_IF;
   "IEC_Timer_0_DB_68".TON(IN := #_w6, PT := T#500MS);
   #_w7 := "IEC_Timer_0_DB_68".Q AND NOT "AUXILIARY".pulse2[1];   // rising edge
   "AUXILIARY".pulse2[1] := "IEC_Timer_0_DB_68".Q;
   IF #_w7 THEN "trigger2" := TRUE; END_IF;
   #_w8 := "AlwaysTRUE" AND ("BUFF".PROCESS = 97);
   IF #_w8 THEN "REVAMP".L15 := '    VACUUM HOLD END PRESSURE:-'; END_IF;
   "IEC_Timer_0_DB_70".TON(IN := #_w8, PT := T#500MS);
   #_w9 := "IEC_Timer_0_DB_70".Q AND NOT "AUXILIARY".pulse2[2];   // rising edge
   "AUXILIARY".pulse2[2] := "IEC_Timer_0_DB_70".Q;
   IF #_w9 THEN "trigger2" := TRUE; END_IF;
   #_w10 := "AlwaysTRUE" AND ("BUFF".PROCESS = 98);
   IF #_w10 THEN "REVAMP".L15 := '    ACTUAL LEAKAGE:-'; END_IF;
   "IEC_Timer_0_DB_71".TON(IN := #_w10, PT := T#500MS);
   #_w11 := "IEC_Timer_0_DB_71".Q AND NOT "AUXILIARY".pulse2[3];   // rising edge
   "AUXILIARY".pulse2[3] := "IEC_Timer_0_DB_71".Q;
   IF #_w11 THEN "trigger2" := TRUE; END_IF;
   #_w12 := "AlwaysTRUE" AND ("BUFF".PROCESS = 99);
   IF #_w12 THEN "REVAMP".L15 := '    ACCEPTANCE LEAKAGE:-'; END_IF;
   "IEC_Timer_0_DB_72".TON(IN := #_w12, PT := T#500MS);
   #_w13 := "IEC_Timer_0_DB_72".Q AND NOT "AUXILIARY".pulse2[4];   // rising edge
   "AUXILIARY".pulse2[4] := "IEC_Timer_0_DB_72".Q;
   IF #_w13 THEN "trigger2" := TRUE; END_IF;
   #_w14 := "AlwaysTRUE" AND ("BUFF".PROCESS = 100);
   #_w15 := #_w14 AND ("VCC DIFF" <= "RETAIN"."SET ACCEPTANCE LEAK");
   IF #_w15 THEN "REVAMP".L15 := '     RESULT:- VACUUM LEAK TEST PASS            '; END_IF;
   "IEC_Timer_0_DB_73".TON(IN := #_w15, PT := T#500MS);
   #_w16 := "IEC_Timer_0_DB_73".Q AND NOT "AUXILIARY".pulse2[5];   // rising edge
   "AUXILIARY".pulse2[5] := "IEC_Timer_0_DB_73".Q;
   IF #_w16 THEN "trigger2" := TRUE; END_IF;
   #_w17 := #_w14 AND ("VCC DIFF" > "RETAIN"."SET ACCEPTANCE LEAK");
   IF #_w17 THEN "REVAMP".L15 := '    RESULT:- VACUUM LEAK TEST FAIL                   '; END_IF;
   "IEC_Timer_0_DB_74".TON(IN := #_w17, PT := T#500MS);
   #_w18 := "IEC_Timer_0_DB_74".Q AND NOT "AUXILIARY".pulse2[6];   // rising edge
   "AUXILIARY".pulse2[6] := "IEC_Timer_0_DB_74".Q;
   IF #_w18 THEN "trigger2" := TRUE; END_IF;
   IF "IEC_Timer_0_DB_74".Q THEN "VACCUM FAIL" := TRUE; END_IF;
   #_w19 := "AlwaysTRUE" AND ("BUFF".PROCESS = 101);
   IF #_w19 THEN "REVAMP".L15 := '     '; END_IF;
   "IEC_Timer_0_DB_54".TON(IN := #_w19, PT := T#3s);
   IF "IEC_Timer_0_DB_54".Q THEN
       "BUFF".PROCESS := 102;
       "trigger2" := TRUE;
   END_IF;
   #_w20 := "AlwaysTRUE" AND ("BUFF".PROCESS = 102);
   "IEC_Timer_0_DB_75".TON(IN := #_w20, PT := T#2S);
   IF "IEC_Timer_0_DB_75".Q THEN
       "BUFF".PROCESS := 0;
       "CYCLE END" := TRUE;
       "IO BITS".HOOTER := TRUE;
   END_IF;
   "VACUUM DONE" := #_w20;
   IF "AlwaysTRUE" AND ("BUFF".PROCESS <> 100) THEN "VACCUM FAIL" := FALSE; END_IF;
END_REGION

REGION Network 7
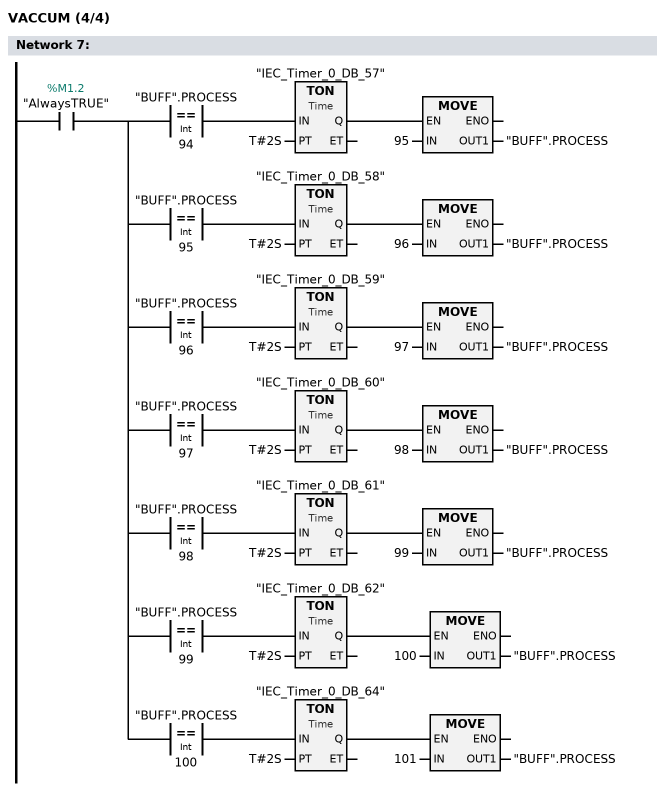
   RUNG wire#powerrail
      Contact( "AlwaysTRUE" )
      wire#w1
      { S7_Templates := "SrcType := Int" } EQ_Contact(in1 := "BUFF".PROCESS, in2 := 94)
      { S7_Templates := "time_type := Time" } "IEC_Timer_0_DB_57".TON(pt := T#2S, et =>)
      Move(in := 95, out1 => "BUFF".PROCESS)
   END_RUNG
   RUNG wire#w1
      { S7_Templates := "SrcType := Int" } EQ_Contact(in1 := "BUFF".PROCESS, in2 := 95)
      { S7_Templates := "time_type := Time" } "IEC_Timer_0_DB_58".TON(pt := T#2S, et =>)
      Move(in := 96, out1 => "BUFF".PROCESS)
   END_RUNG
   RUNG wire#w1
      { S7_Templates := "SrcType := Int" } EQ_Contact(in1 := "BUFF".PROCESS, in2 := 96)
      { S7_Templates := "time_type := Time" } "IEC_Timer_0_DB_59".TON(pt := T#2S, et =>)
      Move(in := 97, out1 => "BUFF".PROCESS)
   END_RUNG
   RUNG wire#w1
      { S7_Templates := "SrcType := Int" } EQ_Contact(in1 := "BUFF".PROCESS, in2 := 97)
      { S7_Templates := "time_type := Time" } "IEC_Timer_0_DB_60".TON(pt := T#2S, et =>)
      Move(in := 98, out1 => "BUFF".PROCESS)
   END_RUNG
   RUNG wire#w1
      { S7_Templates := "SrcType := Int" } EQ_Contact(in1 := "BUFF".PROCESS, in2 := 98)
      { S7_Templates := "time_type := Time" } "IEC_Timer_0_DB_61".TON(pt := T#2S, et =>)
      Move(in := 99, out1 => "BUFF".PROCESS)
   END_RUNG
   RUNG wire#w1
      { S7_Templates := "SrcType := Int" } EQ_Contact(in1 := "BUFF".PROCESS, in2 := 99)
      { S7_Templates := "time_type := Time" } "IEC_Timer_0_DB_62".TON(pt := T#2S, et =>)
      Move(in := 100, out1 => "BUFF".PROCESS)
   END_RUNG
   RUNG wire#w1
      { S7_Templates := "SrcType := Int" } EQ_Contact(in1 := "BUFF".PROCESS, in2 := 100)
      { S7_Templates := "time_type := Time" } "IEC_Timer_0_DB_64".TON(pt := T#2S, et =>)
      Move(in := 101, out1 => "BUFF".PROCESS)
   END_RUNG
   // the same network as SCL:
   "IEC_Timer_0_DB_57".TON(IN := "AlwaysTRUE" AND ("BUFF".PROCESS = 94), PT := T#2S);
   IF "IEC_Timer_0_DB_57".Q THEN "BUFF".PROCESS := 95; END_IF;
   "IEC_Timer_0_DB_58".TON(IN := "AlwaysTRUE" AND ("BUFF".PROCESS = 95), PT := T#2S);
   IF "IEC_Timer_0_DB_58".Q THEN "BUFF".PROCESS := 96; END_IF;
   "IEC_Timer_0_DB_59".TON(IN := "AlwaysTRUE" AND ("BUFF".PROCESS = 96), PT := T#2S);
   IF "IEC_Timer_0_DB_59".Q THEN "BUFF".PROCESS := 97; END_IF;
   "IEC_Timer_0_DB_60".TON(IN := "AlwaysTRUE" AND ("BUFF".PROCESS = 97), PT := T#2S);
   IF "IEC_Timer_0_DB_60".Q THEN "BUFF".PROCESS := 98; END_IF;
   "IEC_Timer_0_DB_61".TON(IN := "AlwaysTRUE" AND ("BUFF".PROCESS = 98), PT := T#2S);
   IF "IEC_Timer_0_DB_61".Q THEN "BUFF".PROCESS := 99; END_IF;
   "IEC_Timer_0_DB_62".TON(IN := "AlwaysTRUE" AND ("BUFF".PROCESS = 99), PT := T#2S);
   IF "IEC_Timer_0_DB_62".Q THEN "BUFF".PROCESS := 100; END_IF;
   "IEC_Timer_0_DB_64".TON(IN := "AlwaysTRUE" AND ("BUFF".PROCESS = 100), PT := T#2S);
   IF "IEC_Timer_0_DB_64".Q THEN "BUFF".PROCESS := 101; END_IF;
END_REGION
END_FUNCTION

FUNCTION "CPEC" : Void   // FC17, LAD
{ S7_Optimized_Access := 'TRUE' }
// stored: SetENOAutomatically false
   VAR_TEMP   // added for the SCL form of the ladder/FBD networks
      _w1 : Bool;
      _w2 : Bool;
      _w3 : Bool;
      _w4 : Bool;
      _w5 : Bool;
      _w6 : Bool;
      _w7 : Bool;
      _w8 : Bool;
      _w9 : Bool;
      _w10 : Bool;
      _w11 : Bool;
      _w12 : Bool;
      _w13 : Bool;
      _w14 : Bool;
      _w15 : Bool;
      _w16 : Bool;
      _w17 : Bool;
      _w18 : Bool;
      _w19 : Bool;
      _w20 : Bool;
      _w21 : Bool;
      _w22 : Bool;
      _w23 : Bool;
      _w24 : Bool;
      _w25 : Bool;
      _w26 : Bool;
      _w27 : Bool;
      _w28 : Bool;
      _w29 : Bool;
      _w30 : Bool;
      _w31 : Bool;
      _w32 : Bool;
      _w33 : Bool;
      _w34 : Bool;
      _w35 : Bool;
      _w36 : Bool;
      _w37 : Bool;
      _w38 : Bool;
      _w39 : Bool;
      _w40 : Bool;
      _w41 : Bool;
      _w42 : Bool;
      _w43 : Bool;
      _w44 : Bool;
      _w45 : Bool;
      _w46 : Bool;
      _w47 : Bool;
      _w48 : Bool;
      _w49 : Bool;
      _w50 : Bool;
      _w51 : Bool;
      _w52 : Bool;
      _w53 : Bool;
      _w54 : Bool;
   END_VAR
BEGIN

REGION Network 1
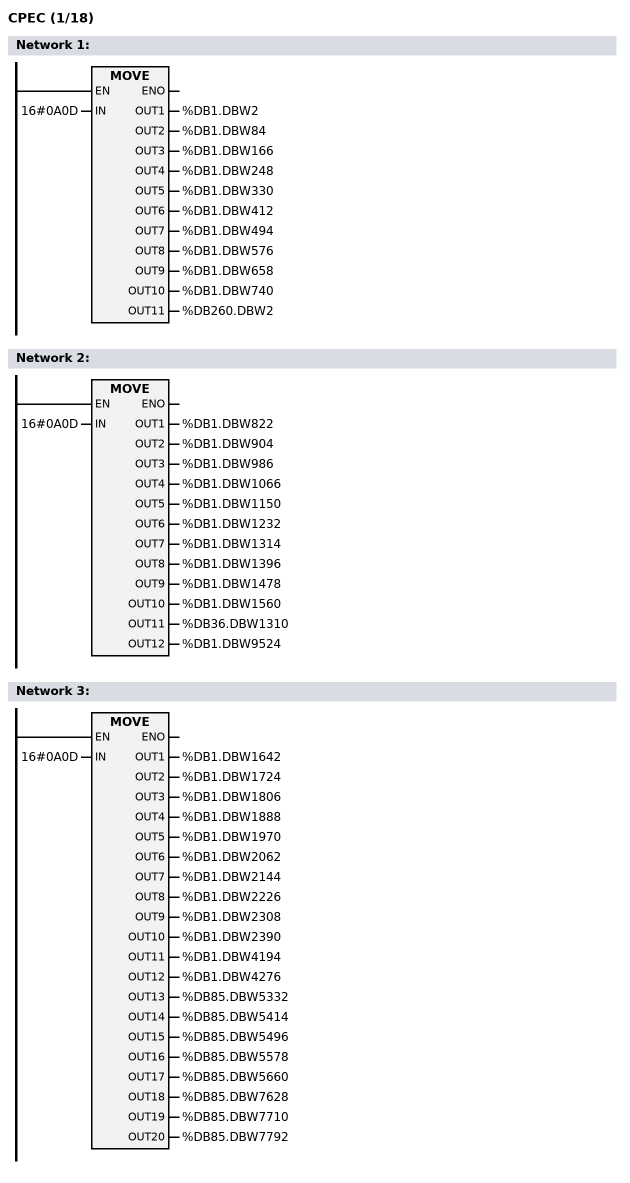
   RUNG wire#powerrail
      Move(in := 16#0A0D, out1 => %DB1.DBW2, out2 => %DB1.DBW84, out3 => %DB1.DBW166, out4 => %DB1.DBW248, out5 => %DB1.DBW330, out6 => %DB1.DBW412, out7 => %DB1.DBW494, out8 => %DB1.DBW576, out9 => %DB1.DBW658, out10 => %DB1.DBW740, out11 => %DB260.DBW2)
   END_RUNG
   // the same network as SCL:
   %DB1.DBW2 := 16#0A0D;
   %DB1.DBW84 := 16#0A0D;
   %DB1.DBW166 := 16#0A0D;
   %DB1.DBW248 := 16#0A0D;
   %DB1.DBW330 := 16#0A0D;
   %DB1.DBW412 := 16#0A0D;
   %DB1.DBW494 := 16#0A0D;
   %DB1.DBW576 := 16#0A0D;
   %DB1.DBW658 := 16#0A0D;
   %DB1.DBW740 := 16#0A0D;
   %DB260.DBW2 := 16#0A0D;
END_REGION

REGION Network 2
   RUNG wire#powerrail
      Move(in := 16#0A0D, out1 => %DB1.DBW822, out2 => %DB1.DBW904, out3 => %DB1.DBW986, out4 => %DB1.DBW1066, out5 => %DB1.DBW1150, out6 => %DB1.DBW1232, out7 => %DB1.DBW1314, out8 => %DB1.DBW1396, out9 => %DB1.DBW1478, out10 => %DB1.DBW1560, out11 => %DB36.DBW1310, out12 => %DB1.DBW9524)
   END_RUNG
   // the same network as SCL:
   %DB1.DBW822 := 16#0A0D;
   %DB1.DBW904 := 16#0A0D;
   %DB1.DBW986 := 16#0A0D;
   %DB1.DBW1066 := 16#0A0D;
   %DB1.DBW1150 := 16#0A0D;
   %DB1.DBW1232 := 16#0A0D;
   %DB1.DBW1314 := 16#0A0D;
   %DB1.DBW1396 := 16#0A0D;
   %DB1.DBW1478 := 16#0A0D;
   %DB1.DBW1560 := 16#0A0D;
   %DB36.DBW1310 := 16#0A0D;
   %DB1.DBW9524 := 16#0A0D;
END_REGION

REGION Network 3
   RUNG wire#powerrail
      Move(in := 16#0A0D, out1 => %DB1.DBW1642, out2 => %DB1.DBW1724, out3 => %DB1.DBW1806, out4 => %DB1.DBW1888, out5 => %DB1.DBW1970, out6 => %DB1.DBW2062, out7 => %DB1.DBW2144, out8 => %DB1.DBW2226, out9 => %DB1.DBW2308, out10 => %DB1.DBW2390, out11 => %DB1.DBW4194, out12 => %DB1.DBW4276, out13 => %DB85.DBW5332, out14 => %DB85.DBW5414, out15 => %DB85.DBW5496, out16 => %DB85.DBW5578, out17 => %DB85.DBW5660, out18 => %DB85.DBW7628, out19 => %DB85.DBW7710, out20 => %DB85.DBW7792)
   END_RUNG
   // the same network as SCL:
   %DB1.DBW1642 := 16#0A0D;
   %DB1.DBW1724 := 16#0A0D;
   %DB1.DBW1806 := 16#0A0D;
   %DB1.DBW1888 := 16#0A0D;
   %DB1.DBW1970 := 16#0A0D;
   %DB1.DBW2062 := 16#0A0D;
   %DB1.DBW2144 := 16#0A0D;
   %DB1.DBW2226 := 16#0A0D;
   %DB1.DBW2308 := 16#0A0D;
   %DB1.DBW2390 := 16#0A0D;
   %DB1.DBW4194 := 16#0A0D;
   %DB1.DBW4276 := 16#0A0D;
   %DB85.DBW5332 := 16#0A0D;
   %DB85.DBW5414 := 16#0A0D;
   %DB85.DBW5496 := 16#0A0D;
   %DB85.DBW5578 := 16#0A0D;
   %DB85.DBW5660 := 16#0A0D;
   %DB85.DBW7628 := 16#0A0D;
   %DB85.DBW7710 := 16#0A0D;
   %DB85.DBW7792 := 16#0A0D;
END_REGION

REGION Network 4
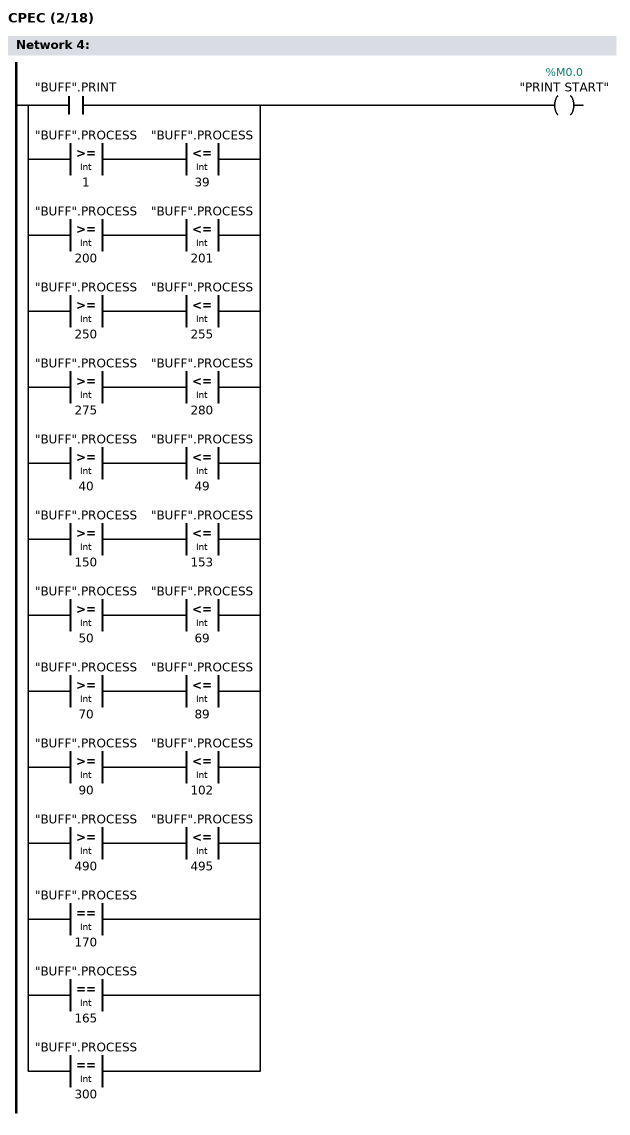
   RUNG wire#powerrail
      Contact( "BUFF".PRINT )
      wire#w1
      Coil( "PRINT START" )
   END_RUNG
   RUNG wire#powerrail
      { S7_Templates := "SrcType := Int" } GE_Contact(in1 := "BUFF".PROCESS, in2 := 1)
      { S7_Templates := "SrcType := Int" } LE_Contact(in1 := "BUFF".PROCESS, in2 := 39)
   END_RUNG wire#w1
   RUNG wire#powerrail
      { S7_Templates := "SrcType := Int" } GE_Contact(in1 := "BUFF".PROCESS, in2 := 200)
      { S7_Templates := "SrcType := Int" } LE_Contact(in1 := "BUFF".PROCESS, in2 := 201)
   END_RUNG wire#w1
   RUNG wire#powerrail
      { S7_Templates := "SrcType := Int" } GE_Contact(in1 := "BUFF".PROCESS, in2 := 250)
      { S7_Templates := "SrcType := Int" } LE_Contact(in1 := "BUFF".PROCESS, in2 := 255)
   END_RUNG wire#w1
   RUNG wire#powerrail
      { S7_Templates := "SrcType := Int" } GE_Contact(in1 := "BUFF".PROCESS, in2 := 275)
      { S7_Templates := "SrcType := Int" } LE_Contact(in1 := "BUFF".PROCESS, in2 := 280)
   END_RUNG wire#w1
   RUNG wire#powerrail
      { S7_Templates := "SrcType := Int" } GE_Contact(in1 := "BUFF".PROCESS, in2 := 40)
      { S7_Templates := "SrcType := Int" } LE_Contact(in1 := "BUFF".PROCESS, in2 := 49)
   END_RUNG wire#w1
   RUNG wire#powerrail
      { S7_Templates := "SrcType := Int" } GE_Contact(in1 := "BUFF".PROCESS, in2 := 150)
      { S7_Templates := "SrcType := Int" } LE_Contact(in1 := "BUFF".PROCESS, in2 := 153)
   END_RUNG wire#w1
   RUNG wire#powerrail
      { S7_Templates := "SrcType := Int" } GE_Contact(in1 := "BUFF".PROCESS, in2 := 50)
      { S7_Templates := "SrcType := Int" } LE_Contact(in1 := "BUFF".PROCESS, in2 := 69)
   END_RUNG wire#w1
   RUNG wire#powerrail
      { S7_Templates := "SrcType := Int" } GE_Contact(in1 := "BUFF".PROCESS, in2 := 70)
      { S7_Templates := "SrcType := Int" } LE_Contact(in1 := "BUFF".PROCESS, in2 := 89)
   END_RUNG wire#w1
   RUNG wire#powerrail
      { S7_Templates := "SrcType := Int" } GE_Contact(in1 := "BUFF".PROCESS, in2 := 90)
      { S7_Templates := "SrcType := Int" } LE_Contact(in1 := "BUFF".PROCESS, in2 := 102)
   END_RUNG wire#w1
   RUNG wire#powerrail
      { S7_Templates := "SrcType := Int" } GE_Contact(in1 := "BUFF".PROCESS, in2 := 490)
      { S7_Templates := "SrcType := Int" } LE_Contact(in1 := "BUFF".PROCESS, in2 := 495)
   END_RUNG wire#w1
   RUNG wire#powerrail
      { S7_Templates := "SrcType := Int" } EQ_Contact(in1 := "BUFF".PROCESS, in2 := 170)
   END_RUNG wire#w1
   RUNG wire#powerrail
      { S7_Templates := "SrcType := Int" } EQ_Contact(in1 := "BUFF".PROCESS, in2 := 165)
   END_RUNG wire#w1
   RUNG wire#powerrail
      { S7_Templates := "SrcType := Int" } EQ_Contact(in1 := "BUFF".PROCESS, in2 := 300)
   END_RUNG wire#w1
   // the same network as SCL:
   "PRINT START" := "BUFF".PRINT OR (("BUFF".PROCESS >= 1) AND ("BUFF".PROCESS <= 39)) OR (("BUFF".PROCESS >= 200) AND ("BUFF".PROCESS <= 201)) OR (("BUFF".PROCESS >= 250) AND ("BUFF".PROCESS <= 255)) OR (("BUFF".PROCESS >= 275) AND ("BUFF".PROCESS <= 280)) OR (("BUFF".PROCESS >= 40) AND ("BUFF".PROCESS <= 49)) OR (("BUFF".PROCESS >= 150) AND ("BUFF".PROCESS <= 153)) OR (("BUFF".PROCESS >= 50) AND ("BUFF".PROCESS <= 69)) OR (("BUFF".PROCESS >= 70) AND ("BUFF".PROCESS <= 89)) OR (("BUFF".PROCESS >= 90) AND ("BUFF".PROCESS <= 102)) OR (("BUFF".PROCESS >= 490) AND ("BUFF".PROCESS <= 495)) OR ("BUFF".PROCESS = 170) OR ("BUFF".PROCESS = 165) OR ("BUFF".PROCESS = 300);
END_REGION

REGION Network 5
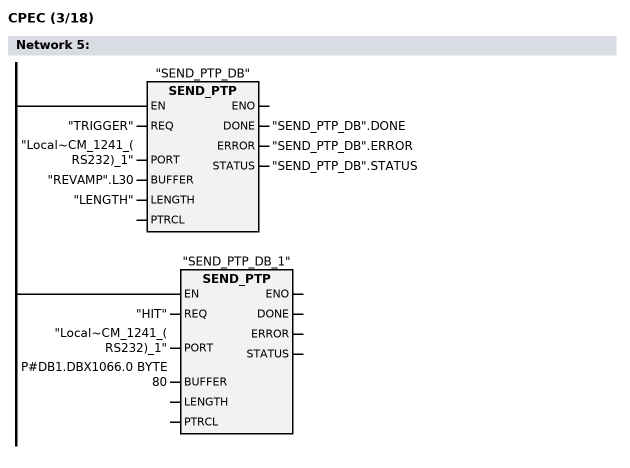
   RUNG wire#powerrail
      "SEND_PTP_DB".SEND_PTP(REQ := "TRIGGER", PORT := "Local~CM_1241_(RS232)_1", BUFFER := "REVAMP".L30, LENGTH := "LENGTH", PTRCL :=, DONE => "SEND_PTP_DB".DONE, ERROR => "SEND_PTP_DB".ERROR, STATUS => "SEND_PTP_DB".STATUS)
   END_RUNG
   RUNG wire#powerrail
      "SEND_PTP_DB_1".SEND_PTP(REQ := "HIT", PORT := "Local~CM_1241_(RS232)_1", BUFFER := P#DB1.DBX1066.0 BYTE 80, LENGTH :=, PTRCL :=, DONE =>, ERROR =>, STATUS =>)
   END_RUNG
   // the same network as SCL:
   "SEND_PTP_DB"(REQ := "TRIGGER",   // SEND_PTP
                 PORT := "Local~CM_1241_(RS232)_1",
                 BUFFER := "REVAMP".L30,
                 LENGTH := "LENGTH",
                 DONE => "SEND_PTP_DB".DONE,
                 ERROR => "SEND_PTP_DB".ERROR,
                 STATUS => "SEND_PTP_DB".STATUS);
   "SEND_PTP_DB_1"(REQ := "HIT", PORT := "Local~CM_1241_(RS232)_1", BUFFER := P#DB1.DBX1066.0 BYTE 80);   // SEND_PTP
END_REGION

REGION Network 6
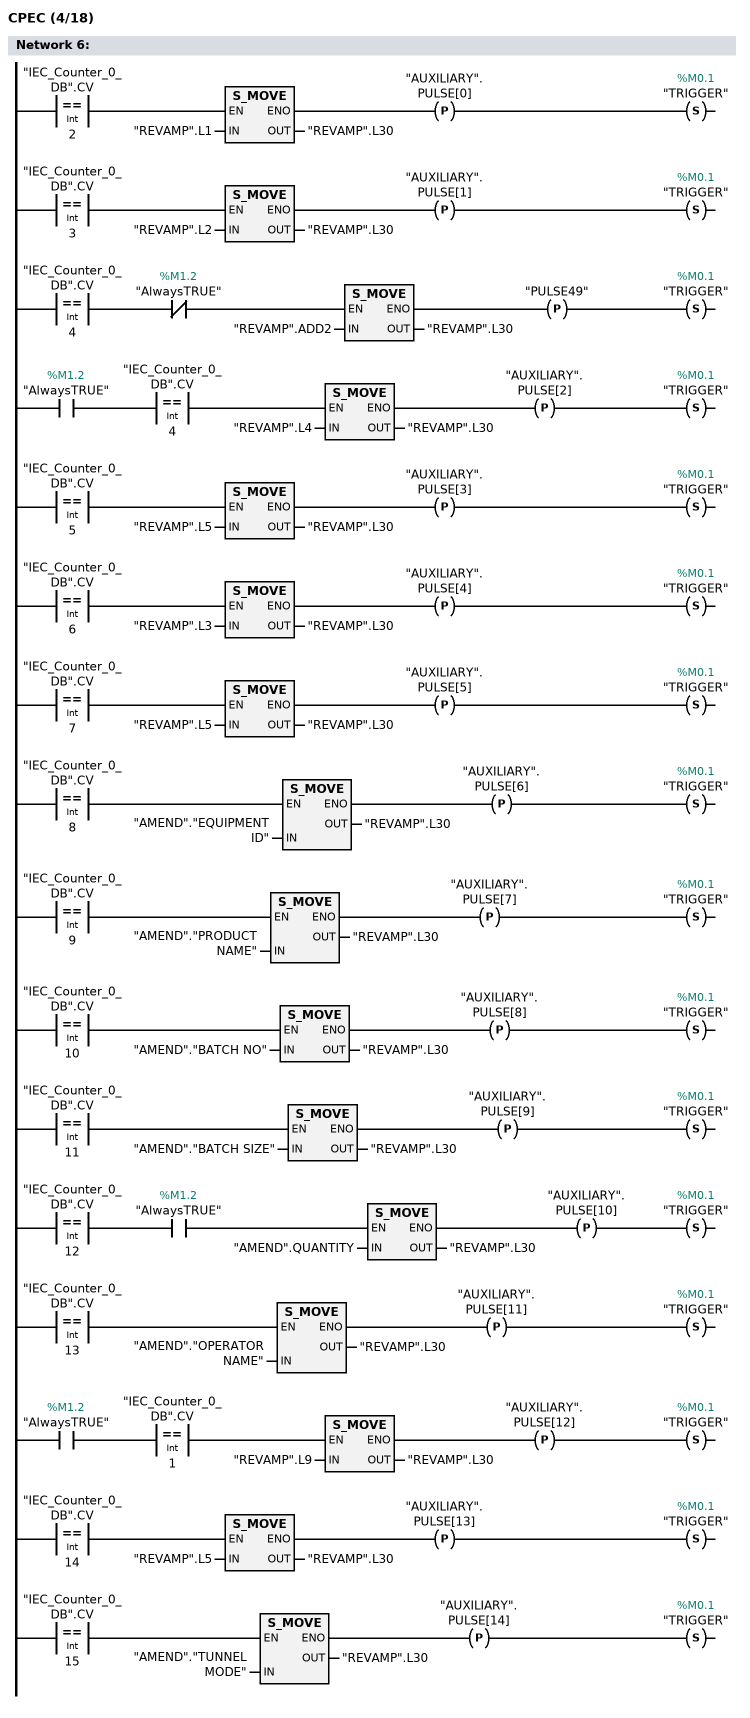
   RUNG wire#powerrail
      { S7_Templates := "SrcType := Int" } EQ_Contact(in1 := "IEC_Counter_0_DB".CV, in2 := 2)
      S_Move(in := "REVAMP".L1, out => "REVAMP".L30)
      P_Trig( "AUXILIARY".PULSE[0] )
      S_Coil( "TRIGGER" )
   END_RUNG
   RUNG wire#powerrail
      { S7_Templates := "SrcType := Int" } EQ_Contact(in1 := "IEC_Counter_0_DB".CV, in2 := 3)
      S_Move(in := "REVAMP".L2, out => "REVAMP".L30)
      P_Trig( "AUXILIARY".PULSE[1] )
      S_Coil( "TRIGGER" )
   END_RUNG
   RUNG wire#powerrail
      { S7_Templates := "SrcType := Int" } EQ_Contact(in1 := "IEC_Counter_0_DB".CV, in2 := 4)
      I_Contact( "AlwaysTRUE" )
      S_Move(in := "REVAMP".ADD2, out => "REVAMP".L30)
      P_Trig( "PULSE49" )
      S_Coil( "TRIGGER" )
   END_RUNG
   RUNG wire#powerrail
      Contact( "AlwaysTRUE" )
      { S7_Templates := "SrcType := Int" } EQ_Contact(in1 := "IEC_Counter_0_DB".CV, in2 := 4)
      S_Move(in := "REVAMP".L4, out => "REVAMP".L30)
      P_Trig( "AUXILIARY".PULSE[2] )
      S_Coil( "TRIGGER" )
   END_RUNG
   RUNG wire#powerrail
      { S7_Templates := "SrcType := Int" } EQ_Contact(in1 := "IEC_Counter_0_DB".CV, in2 := 5)
      S_Move(in := "REVAMP".L5, out => "REVAMP".L30)
      P_Trig( "AUXILIARY".PULSE[3] )
      S_Coil( "TRIGGER" )
   END_RUNG
   RUNG wire#powerrail
      { S7_Templates := "SrcType := Int" } EQ_Contact(in1 := "IEC_Counter_0_DB".CV, in2 := 6)
      S_Move(in := "REVAMP".L3, out => "REVAMP".L30)
      P_Trig( "AUXILIARY".PULSE[4] )
      S_Coil( "TRIGGER" )
   END_RUNG
   RUNG wire#powerrail
      { S7_Templates := "SrcType := Int" } EQ_Contact(in1 := "IEC_Counter_0_DB".CV, in2 := 7)
      S_Move(in := "REVAMP".L5, out => "REVAMP".L30)
      P_Trig( "AUXILIARY".PULSE[5] )
      S_Coil( "TRIGGER" )
   END_RUNG
   RUNG wire#powerrail
      { S7_Templates := "SrcType := Int" } EQ_Contact(in1 := "IEC_Counter_0_DB".CV, in2 := 8)
      S_Move(in := "AMEND"."EQUIPMENT ID", out => "REVAMP".L30)
      P_Trig( "AUXILIARY".PULSE[6] )
      S_Coil( "TRIGGER" )
   END_RUNG
   RUNG wire#powerrail
      { S7_Templates := "SrcType := Int" } EQ_Contact(in1 := "IEC_Counter_0_DB".CV, in2 := 9)
      S_Move(in := "AMEND"."PRODUCT NAME", out => "REVAMP".L30)
      P_Trig( "AUXILIARY".PULSE[7] )
      S_Coil( "TRIGGER" )
   END_RUNG
   RUNG wire#powerrail
      { S7_Templates := "SrcType := Int" } EQ_Contact(in1 := "IEC_Counter_0_DB".CV, in2 := 10)
      S_Move(in := "AMEND"."BATCH NO", out => "REVAMP".L30)
      P_Trig( "AUXILIARY".PULSE[8] )
      S_Coil( "TRIGGER" )
   END_RUNG
   RUNG wire#powerrail
      { S7_Templates := "SrcType := Int" } EQ_Contact(in1 := "IEC_Counter_0_DB".CV, in2 := 11)
      S_Move(in := "AMEND"."BATCH SIZE", out => "REVAMP".L30)
      P_Trig( "AUXILIARY".PULSE[9] )
      S_Coil( "TRIGGER" )
   END_RUNG
   RUNG wire#powerrail
      { S7_Templates := "SrcType := Int" } EQ_Contact(in1 := "IEC_Counter_0_DB".CV, in2 := 12)
      Contact( "AlwaysTRUE" )
      S_Move(in := "AMEND".QUANTITY, out => "REVAMP".L30)
      P_Trig( "AUXILIARY".PULSE[10] )
      S_Coil( "TRIGGER" )
   END_RUNG
   RUNG wire#powerrail
      { S7_Templates := "SrcType := Int" } EQ_Contact(in1 := "IEC_Counter_0_DB".CV, in2 := 13)
      S_Move(in := "AMEND"."OPERATOR NAME", out => "REVAMP".L30)
      P_Trig( "AUXILIARY".PULSE[11] )
      S_Coil( "TRIGGER" )
   END_RUNG
   RUNG wire#powerrail
      Contact( "AlwaysTRUE" )
      { S7_Templates := "SrcType := Int" } EQ_Contact(in1 := "IEC_Counter_0_DB".CV, in2 := 1)
      S_Move(in := "REVAMP".L9, out => "REVAMP".L30)
      P_Trig( "AUXILIARY".PULSE[12] )
      S_Coil( "TRIGGER" )
   END_RUNG
   RUNG wire#powerrail
      { S7_Templates := "SrcType := Int" } EQ_Contact(in1 := "IEC_Counter_0_DB".CV, in2 := 14)
      S_Move(in := "REVAMP".L5, out => "REVAMP".L30)
      P_Trig( "AUXILIARY".PULSE[13] )
      S_Coil( "TRIGGER" )
   END_RUNG
   RUNG wire#powerrail
      { S7_Templates := "SrcType := Int" } EQ_Contact(in1 := "IEC_Counter_0_DB".CV, in2 := 15)
      S_Move(in := "AMEND"."TUNNEL MODE", out => "REVAMP".L30)
      P_Trig( "AUXILIARY".PULSE[14] )
      S_Coil( "TRIGGER" )
   END_RUNG
   // the same network as SCL:
   #_w1 := "IEC_Counter_0_DB".CV = 2;
   IF #_w1 THEN "REVAMP".L30 := "REVAMP".L1; END_IF;
   #_w2 := #_w1 AND NOT "AUXILIARY".PULSE[0];   // rising edge
   "AUXILIARY".PULSE[0] := #_w1;
   IF #_w2 THEN "TRIGGER" := TRUE; END_IF;
   #_w3 := "IEC_Counter_0_DB".CV = 3;
   IF #_w3 THEN "REVAMP".L30 := "REVAMP".L2; END_IF;
   #_w4 := #_w3 AND NOT "AUXILIARY".PULSE[1];   // rising edge
   "AUXILIARY".PULSE[1] := #_w3;
   IF #_w4 THEN "TRIGGER" := TRUE; END_IF;
   #_w5 := ("IEC_Counter_0_DB".CV = 4) AND NOT "AlwaysTRUE";
   IF #_w5 THEN "REVAMP".L30 := "REVAMP".ADD2; END_IF;
   #_w6 := #_w5 AND NOT "PULSE49";   // rising edge
   "PULSE49" := #_w5;
   IF #_w6 THEN "TRIGGER" := TRUE; END_IF;
   #_w7 := "AlwaysTRUE" AND ("IEC_Counter_0_DB".CV = 4);
   IF #_w7 THEN "REVAMP".L30 := "REVAMP".L4; END_IF;
   #_w8 := #_w7 AND NOT "AUXILIARY".PULSE[2];   // rising edge
   "AUXILIARY".PULSE[2] := #_w7;
   IF #_w8 THEN "TRIGGER" := TRUE; END_IF;
   #_w9 := "IEC_Counter_0_DB".CV = 5;
   IF #_w9 THEN "REVAMP".L30 := "REVAMP".L5; END_IF;
   #_w10 := #_w9 AND NOT "AUXILIARY".PULSE[3];   // rising edge
   "AUXILIARY".PULSE[3] := #_w9;
   IF #_w10 THEN "TRIGGER" := TRUE; END_IF;
   #_w11 := "IEC_Counter_0_DB".CV = 6;
   IF #_w11 THEN "REVAMP".L30 := "REVAMP".L3; END_IF;
   #_w12 := #_w11 AND NOT "AUXILIARY".PULSE[4];   // rising edge
   "AUXILIARY".PULSE[4] := #_w11;
   IF #_w12 THEN "TRIGGER" := TRUE; END_IF;
   #_w13 := "IEC_Counter_0_DB".CV = 7;
   IF #_w13 THEN "REVAMP".L30 := "REVAMP".L5; END_IF;
   #_w14 := #_w13 AND NOT "AUXILIARY".PULSE[5];   // rising edge
   "AUXILIARY".PULSE[5] := #_w13;
   IF #_w14 THEN "TRIGGER" := TRUE; END_IF;
   #_w15 := "IEC_Counter_0_DB".CV = 8;
   IF #_w15 THEN "REVAMP".L30 := "AMEND"."EQUIPMENT ID"; END_IF;
   #_w16 := #_w15 AND NOT "AUXILIARY".PULSE[6];   // rising edge
   "AUXILIARY".PULSE[6] := #_w15;
   IF #_w16 THEN "TRIGGER" := TRUE; END_IF;
   #_w17 := "IEC_Counter_0_DB".CV = 9;
   IF #_w17 THEN "REVAMP".L30 := "AMEND"."PRODUCT NAME"; END_IF;
   #_w18 := #_w17 AND NOT "AUXILIARY".PULSE[7];   // rising edge
   "AUXILIARY".PULSE[7] := #_w17;
   IF #_w18 THEN "TRIGGER" := TRUE; END_IF;
   #_w19 := "IEC_Counter_0_DB".CV = 10;
   IF #_w19 THEN "REVAMP".L30 := "AMEND"."BATCH NO"; END_IF;
   #_w20 := #_w19 AND NOT "AUXILIARY".PULSE[8];   // rising edge
   "AUXILIARY".PULSE[8] := #_w19;
   IF #_w20 THEN "TRIGGER" := TRUE; END_IF;
   #_w21 := "IEC_Counter_0_DB".CV = 11;
   IF #_w21 THEN "REVAMP".L30 := "AMEND"."BATCH SIZE"; END_IF;
   #_w22 := #_w21 AND NOT "AUXILIARY".PULSE[9];   // rising edge
   "AUXILIARY".PULSE[9] := #_w21;
   IF #_w22 THEN "TRIGGER" := TRUE; END_IF;
   #_w23 := ("IEC_Counter_0_DB".CV = 12) AND "AlwaysTRUE";
   IF #_w23 THEN "REVAMP".L30 := "AMEND".QUANTITY; END_IF;
   #_w24 := #_w23 AND NOT "AUXILIARY".PULSE[10];   // rising edge
   "AUXILIARY".PULSE[10] := #_w23;
   IF #_w24 THEN "TRIGGER" := TRUE; END_IF;
   #_w25 := "IEC_Counter_0_DB".CV = 13;
   IF #_w25 THEN "REVAMP".L30 := "AMEND"."OPERATOR NAME"; END_IF;
   #_w26 := #_w25 AND NOT "AUXILIARY".PULSE[11];   // rising edge
   "AUXILIARY".PULSE[11] := #_w25;
   IF #_w26 THEN "TRIGGER" := TRUE; END_IF;
   #_w27 := "AlwaysTRUE" AND ("IEC_Counter_0_DB".CV = 1);
   IF #_w27 THEN "REVAMP".L30 := "REVAMP".L9; END_IF;
   #_w28 := #_w27 AND NOT "AUXILIARY".PULSE[12];   // rising edge
   "AUXILIARY".PULSE[12] := #_w27;
   IF #_w28 THEN "TRIGGER" := TRUE; END_IF;
   #_w29 := "IEC_Counter_0_DB".CV = 14;
   IF #_w29 THEN "REVAMP".L30 := "REVAMP".L5; END_IF;
   #_w30 := #_w29 AND NOT "AUXILIARY".PULSE[13];   // rising edge
   "AUXILIARY".PULSE[13] := #_w29;
   IF #_w30 THEN "TRIGGER" := TRUE; END_IF;
   #_w31 := "IEC_Counter_0_DB".CV = 15;
   IF #_w31 THEN "REVAMP".L30 := "AMEND"."TUNNEL MODE"; END_IF;
   #_w32 := #_w31 AND NOT "AUXILIARY".PULSE[14];   // rising edge
   "AUXILIARY".PULSE[14] := #_w31;
   IF #_w32 THEN "TRIGGER" := TRUE; END_IF;
END_REGION

REGION Network 7
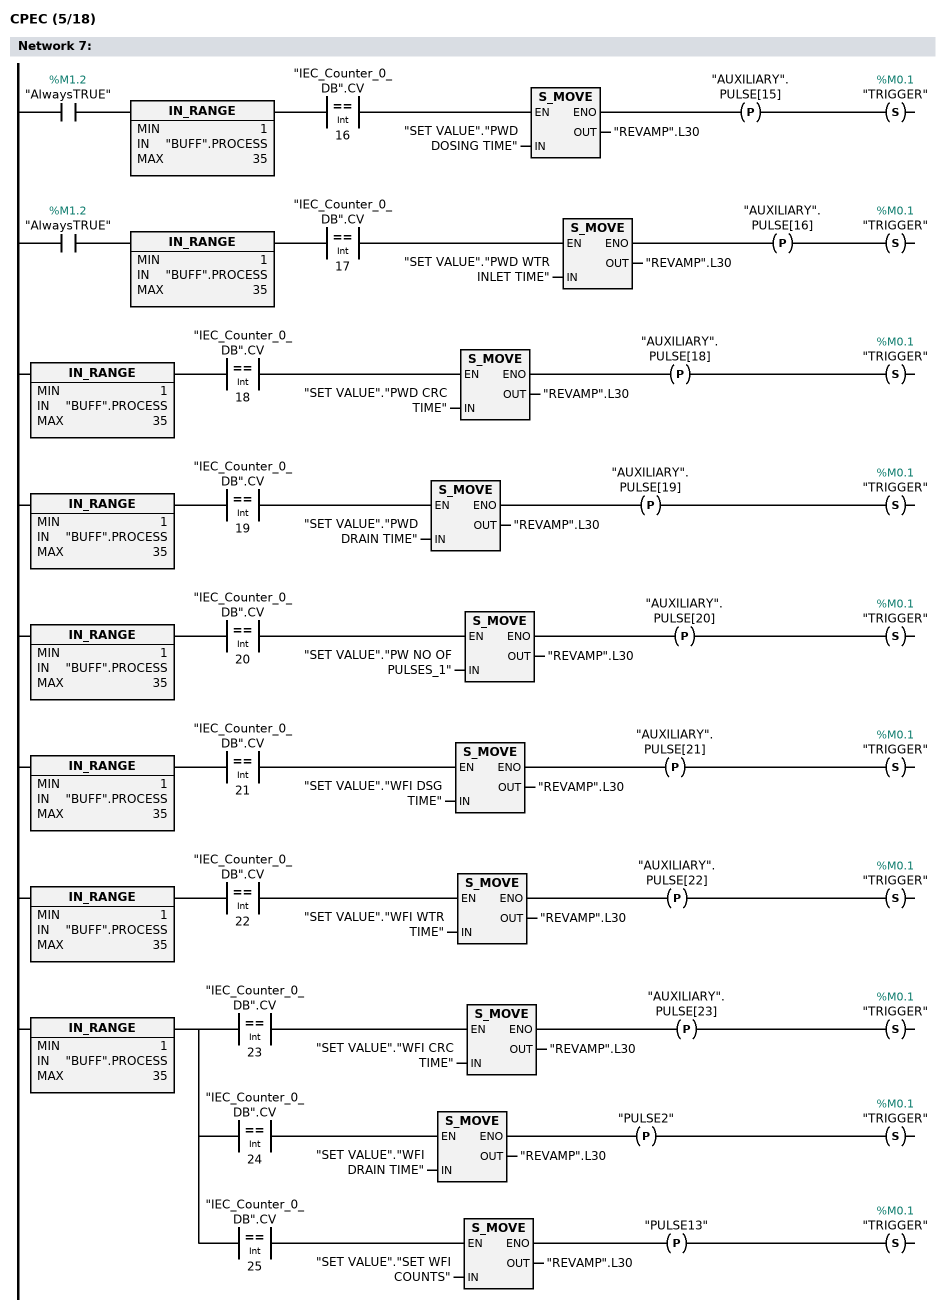
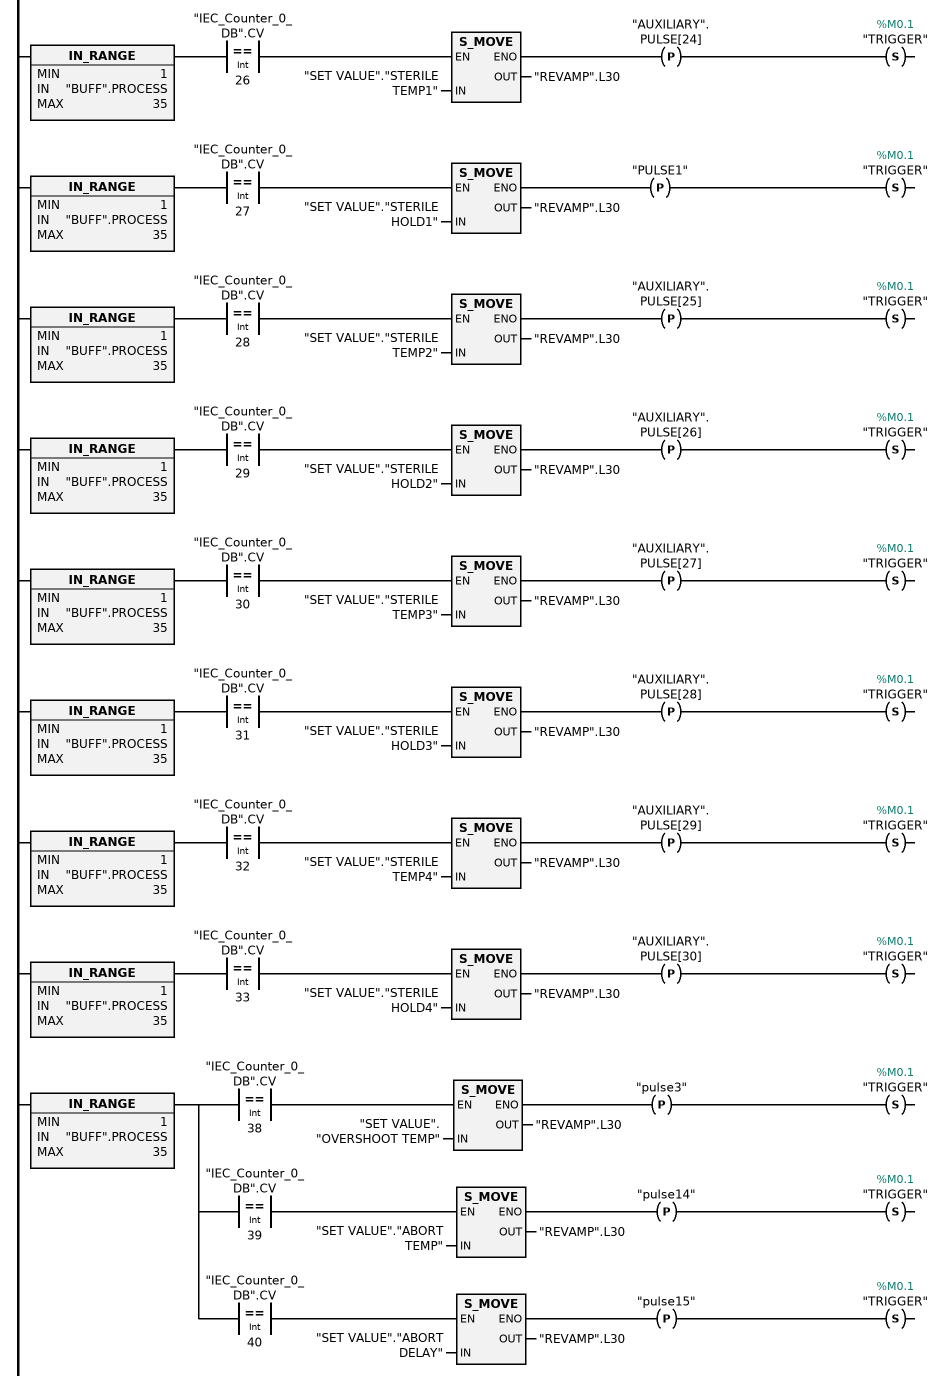
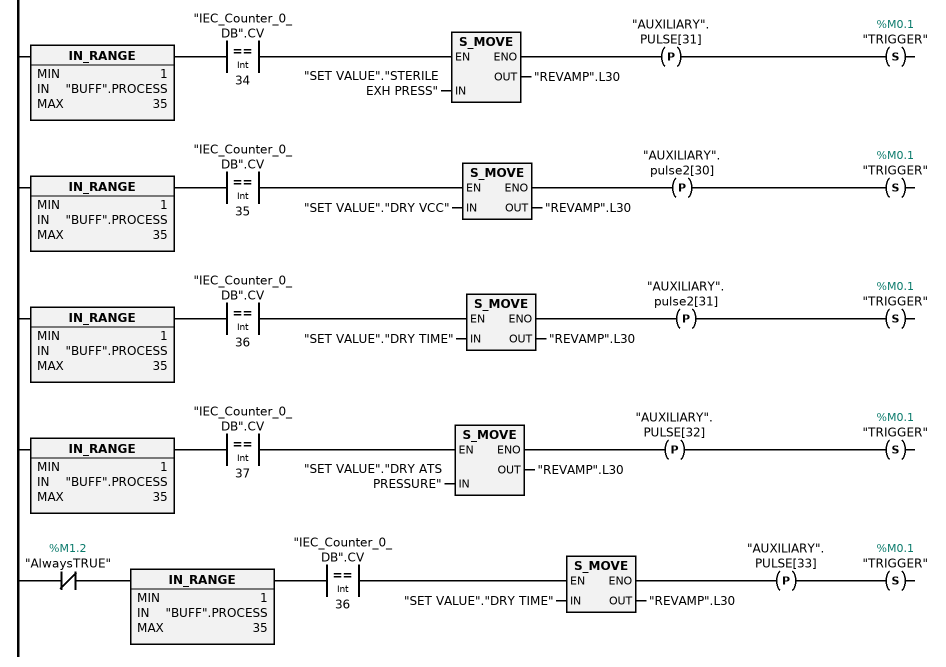
   RUNG wire#powerrail
      Contact( "AlwaysTRUE" )
      { S7_Templates := "SrcType := Int" } InRange(min := 1, in := "BUFF".PROCESS, max := 35)
      { S7_Templates := "SrcType := Int" } EQ_Contact(in1 := "IEC_Counter_0_DB".CV, in2 := 16)
      S_Move(in := "SET VALUE"."PWD DOSING TIME", out => "REVAMP".L30)
      P_Trig( "AUXILIARY".PULSE[15] )
      S_Coil( "TRIGGER" )
   END_RUNG
   RUNG wire#powerrail
      Contact( "AlwaysTRUE" )
      { S7_Templates := "SrcType := Int" } InRange(min := 1, in := "BUFF".PROCESS, max := 35)
      { S7_Templates := "SrcType := Int" } EQ_Contact(in1 := "IEC_Counter_0_DB".CV, in2 := 17)
      S_Move(in := "SET VALUE"."PWD WTR INLET TIME", out => "REVAMP".L30)
      P_Trig( "AUXILIARY".PULSE[16] )
      S_Coil( "TRIGGER" )
   END_RUNG
   RUNG wire#powerrail
      { S7_Templates := "SrcType := Int" } InRange(min := 1, in := "BUFF".PROCESS, max := 35)
      { S7_Templates := "SrcType := Int" } EQ_Contact(in1 := "IEC_Counter_0_DB".CV, in2 := 18)
      S_Move(in := "SET VALUE"."PWD CRC TIME", out => "REVAMP".L30)
      P_Trig( "AUXILIARY".PULSE[18] )
      S_Coil( "TRIGGER" )
   END_RUNG
   RUNG wire#powerrail
      { S7_Templates := "SrcType := Int" } InRange(min := 1, in := "BUFF".PROCESS, max := 35)
      { S7_Templates := "SrcType := Int" } EQ_Contact(in1 := "IEC_Counter_0_DB".CV, in2 := 19)
      S_Move(in := "SET VALUE"."PWD DRAIN TIME", out => "REVAMP".L30)
      P_Trig( "AUXILIARY".PULSE[19] )
      S_Coil( "TRIGGER" )
   END_RUNG
   RUNG wire#powerrail
      { S7_Templates := "SrcType := Int" } InRange(min := 1, in := "BUFF".PROCESS, max := 35)
      { S7_Templates := "SrcType := Int" } EQ_Contact(in1 := "IEC_Counter_0_DB".CV, in2 := 20)
      S_Move(in := "SET VALUE"."PW NO OF PULSES_1", out => "REVAMP".L30)
      P_Trig( "AUXILIARY".PULSE[20] )
      S_Coil( "TRIGGER" )
   END_RUNG
   RUNG wire#powerrail
      { S7_Templates := "SrcType := Int" } InRange(min := 1, in := "BUFF".PROCESS, max := 35)
      { S7_Templates := "SrcType := Int" } EQ_Contact(in1 := "IEC_Counter_0_DB".CV, in2 := 21)
      S_Move(in := "SET VALUE"."WFI DSG TIME", out => "REVAMP".L30)
      P_Trig( "AUXILIARY".PULSE[21] )
      S_Coil( "TRIGGER" )
   END_RUNG
   RUNG wire#powerrail
      { S7_Templates := "SrcType := Int" } InRange(min := 1, in := "BUFF".PROCESS, max := 35)
      { S7_Templates := "SrcType := Int" } EQ_Contact(in1 := "IEC_Counter_0_DB".CV, in2 := 22)
      S_Move(in := "SET VALUE"."WFI WTR TIME", out => "REVAMP".L30)
      P_Trig( "AUXILIARY".PULSE[22] )
      S_Coil( "TRIGGER" )
   END_RUNG
   RUNG wire#powerrail
      { S7_Templates := "SrcType := Int" } InRange(min := 1, in := "BUFF".PROCESS, max := 35)
      wire#w1
      { S7_Templates := "SrcType := Int" } EQ_Contact(in1 := "IEC_Counter_0_DB".CV, in2 := 23)
      S_Move(in := "SET VALUE"."WFI CRC TIME", out => "REVAMP".L30)
      P_Trig( "AUXILIARY".PULSE[23] )
      S_Coil( "TRIGGER" )
   END_RUNG
   RUNG wire#w1
      { S7_Templates := "SrcType := Int" } EQ_Contact(in1 := "IEC_Counter_0_DB".CV, in2 := 24)
      S_Move(in := "SET VALUE"."WFI DRAIN TIME", out => "REVAMP".L30)
      P_Trig( "PULSE2" )
      S_Coil( "TRIGGER" )
   END_RUNG
   RUNG wire#w1
      { S7_Templates := "SrcType := Int" } EQ_Contact(in1 := "IEC_Counter_0_DB".CV, in2 := 25)
      S_Move(in := "SET VALUE"."SET WFI COUNTS", out => "REVAMP".L30)
      P_Trig( "PULSE13" )
      S_Coil( "TRIGGER" )
   END_RUNG
   RUNG wire#powerrail
      { S7_Templates := "SrcType := Int" } InRange(min := 1, in := "BUFF".PROCESS, max := 35)
      { S7_Templates := "SrcType := Int" } EQ_Contact(in1 := "IEC_Counter_0_DB".CV, in2 := 26)
      S_Move(in := "SET VALUE"."STERILE TEMP1", out => "REVAMP".L30)
      P_Trig( "AUXILIARY".PULSE[24] )
      S_Coil( "TRIGGER" )
   END_RUNG
   RUNG wire#powerrail
      { S7_Templates := "SrcType := Int" } InRange(min := 1, in := "BUFF".PROCESS, max := 35)
      { S7_Templates := "SrcType := Int" } EQ_Contact(in1 := "IEC_Counter_0_DB".CV, in2 := 27)
      S_Move(in := "SET VALUE"."STERILE HOLD1", out => "REVAMP".L30)
      P_Trig( "PULSE1" )
      S_Coil( "TRIGGER" )
   END_RUNG
   RUNG wire#powerrail
      { S7_Templates := "SrcType := Int" } InRange(min := 1, in := "BUFF".PROCESS, max := 35)
      { S7_Templates := "SrcType := Int" } EQ_Contact(in1 := "IEC_Counter_0_DB".CV, in2 := 28)
      S_Move(in := "SET VALUE"."STERILE TEMP2", out => "REVAMP".L30)
      P_Trig( "AUXILIARY".PULSE[25] )
      S_Coil( "TRIGGER" )
   END_RUNG
   RUNG wire#powerrail
      { S7_Templates := "SrcType := Int" } InRange(min := 1, in := "BUFF".PROCESS, max := 35)
      { S7_Templates := "SrcType := Int" } EQ_Contact(in1 := "IEC_Counter_0_DB".CV, in2 := 29)
      S_Move(in := "SET VALUE"."STERILE HOLD2", out => "REVAMP".L30)
      P_Trig( "AUXILIARY".PULSE[26] )
      S_Coil( "TRIGGER" )
   END_RUNG
   RUNG wire#powerrail
      { S7_Templates := "SrcType := Int" } InRange(min := 1, in := "BUFF".PROCESS, max := 35)
      { S7_Templates := "SrcType := Int" } EQ_Contact(in1 := "IEC_Counter_0_DB".CV, in2 := 30)
      S_Move(in := "SET VALUE"."STERILE TEMP3", out => "REVAMP".L30)
      P_Trig( "AUXILIARY".PULSE[27] )
      S_Coil( "TRIGGER" )
   END_RUNG
   RUNG wire#powerrail
      { S7_Templates := "SrcType := Int" } InRange(min := 1, in := "BUFF".PROCESS, max := 35)
      { S7_Templates := "SrcType := Int" } EQ_Contact(in1 := "IEC_Counter_0_DB".CV, in2 := 31)
      S_Move(in := "SET VALUE"."STERILE HOLD3", out => "REVAMP".L30)
      P_Trig( "AUXILIARY".PULSE[28] )
      S_Coil( "TRIGGER" )
   END_RUNG
   RUNG wire#powerrail
      { S7_Templates := "SrcType := Int" } InRange(min := 1, in := "BUFF".PROCESS, max := 35)
      { S7_Templates := "SrcType := Int" } EQ_Contact(in1 := "IEC_Counter_0_DB".CV, in2 := 32)
      S_Move(in := "SET VALUE"."STERILE TEMP4", out => "REVAMP".L30)
      P_Trig( "AUXILIARY".PULSE[29] )
      S_Coil( "TRIGGER" )
   END_RUNG
   RUNG wire#powerrail
      { S7_Templates := "SrcType := Int" } InRange(min := 1, in := "BUFF".PROCESS, max := 35)
      { S7_Templates := "SrcType := Int" } EQ_Contact(in1 := "IEC_Counter_0_DB".CV, in2 := 33)
      S_Move(in := "SET VALUE"."STERILE HOLD4", out => "REVAMP".L30)
      P_Trig( "AUXILIARY".PULSE[30] )
      S_Coil( "TRIGGER" )
   END_RUNG
   RUNG wire#powerrail
      { S7_Templates := "SrcType := Int" } InRange(min := 1, in := "BUFF".PROCESS, max := 35)
      wire#w2
      { S7_Templates := "SrcType := Int" } EQ_Contact(in1 := "IEC_Counter_0_DB".CV, in2 := 38)
      S_Move(in := "SET VALUE"."OVERSHOOT TEMP", out => "REVAMP".L30)
      P_Trig( "pulse3" )
      S_Coil( "TRIGGER" )
   END_RUNG
   RUNG wire#w2
      { S7_Templates := "SrcType := Int" } EQ_Contact(in1 := "IEC_Counter_0_DB".CV, in2 := 39)
      S_Move(in := "SET VALUE"."ABORT TEMP", out => "REVAMP".L30)
      P_Trig( "pulse14" )
      S_Coil( "TRIGGER" )
   END_RUNG
   RUNG wire#w2
      { S7_Templates := "SrcType := Int" } EQ_Contact(in1 := "IEC_Counter_0_DB".CV, in2 := 40)
      S_Move(in := "SET VALUE"."ABORT DELAY", out => "REVAMP".L30)
      P_Trig( "pulse15" )
      S_Coil( "TRIGGER" )
   END_RUNG
   RUNG wire#powerrail
      { S7_Templates := "SrcType := Int" } InRange(min := 1, in := "BUFF".PROCESS, max := 35)
      { S7_Templates := "SrcType := Int" } EQ_Contact(in1 := "IEC_Counter_0_DB".CV, in2 := 34)
      S_Move(in := "SET VALUE"."STERILE EXH PRESS", out => "REVAMP".L30)
      P_Trig( "AUXILIARY".PULSE[31] )
      S_Coil( "TRIGGER" )
   END_RUNG
   RUNG wire#powerrail
      { S7_Templates := "SrcType := Int" } InRange(min := 1, in := "BUFF".PROCESS, max := 35)
      { S7_Templates := "SrcType := Int" } EQ_Contact(in1 := "IEC_Counter_0_DB".CV, in2 := 35)
      S_Move(in := "SET VALUE"."DRY VCC", out => "REVAMP".L30)
      P_Trig( "AUXILIARY".pulse2[30] )
      S_Coil( "TRIGGER" )
   END_RUNG
   RUNG wire#powerrail
      { S7_Templates := "SrcType := Int" } InRange(min := 1, in := "BUFF".PROCESS, max := 35)
      { S7_Templates := "SrcType := Int" } EQ_Contact(in1 := "IEC_Counter_0_DB".CV, in2 := 36)
      S_Move(in := "SET VALUE"."DRY TIME", out => "REVAMP".L30)
      P_Trig( "AUXILIARY".pulse2[31] )
      S_Coil( "TRIGGER" )
   END_RUNG
   RUNG wire#powerrail
      { S7_Templates := "SrcType := Int" } InRange(min := 1, in := "BUFF".PROCESS, max := 35)
      { S7_Templates := "SrcType := Int" } EQ_Contact(in1 := "IEC_Counter_0_DB".CV, in2 := 37)
      S_Move(in := "SET VALUE"."DRY ATS PRESSURE", out => "REVAMP".L30)
      P_Trig( "AUXILIARY".PULSE[32] )
      S_Coil( "TRIGGER" )
   END_RUNG
   RUNG wire#powerrail
      I_Contact( "AlwaysTRUE" )
      { S7_Templates := "SrcType := Int" } InRange(min := 1, in := "BUFF".PROCESS, max := 35)
      { S7_Templates := "SrcType := Int" } EQ_Contact(in1 := "IEC_Counter_0_DB".CV, in2 := 36)
      S_Move(in := "SET VALUE"."DRY TIME", out => "REVAMP".L30)
      P_Trig( "AUXILIARY".PULSE[33] )
      S_Coil( "TRIGGER" )
   END_RUNG
   // the same network as SCL:
   #_w1 := "AlwaysTRUE" AND (1 <= "BUFF".PROCESS) AND ("BUFF".PROCESS <= 35) AND ("IEC_Counter_0_DB".CV = 16);
   IF #_w1 THEN "REVAMP".L30 := "SET VALUE"."PWD DOSING TIME"; END_IF;
   #_w2 := #_w1 AND NOT "AUXILIARY".PULSE[15];   // rising edge
   "AUXILIARY".PULSE[15] := #_w1;
   IF #_w2 THEN "TRIGGER" := TRUE; END_IF;
   #_w3 := "AlwaysTRUE" AND (1 <= "BUFF".PROCESS) AND ("BUFF".PROCESS <= 35) AND ("IEC_Counter_0_DB".CV = 17);
   IF #_w3 THEN "REVAMP".L30 := "SET VALUE"."PWD WTR INLET TIME"; END_IF;
   #_w4 := #_w3 AND NOT "AUXILIARY".PULSE[16];   // rising edge
   "AUXILIARY".PULSE[16] := #_w3;
   IF #_w4 THEN "TRIGGER" := TRUE; END_IF;
   #_w5 := (1 <= "BUFF".PROCESS) AND ("BUFF".PROCESS <= 35) AND ("IEC_Counter_0_DB".CV = 18);
   IF #_w5 THEN "REVAMP".L30 := "SET VALUE"."PWD CRC TIME"; END_IF;
   #_w6 := #_w5 AND NOT "AUXILIARY".PULSE[18];   // rising edge
   "AUXILIARY".PULSE[18] := #_w5;
   IF #_w6 THEN "TRIGGER" := TRUE; END_IF;
   #_w7 := (1 <= "BUFF".PROCESS) AND ("BUFF".PROCESS <= 35) AND ("IEC_Counter_0_DB".CV = 19);
   IF #_w7 THEN "REVAMP".L30 := "SET VALUE"."PWD DRAIN TIME"; END_IF;
   #_w8 := #_w7 AND NOT "AUXILIARY".PULSE[19];   // rising edge
   "AUXILIARY".PULSE[19] := #_w7;
   IF #_w8 THEN "TRIGGER" := TRUE; END_IF;
   #_w9 := (1 <= "BUFF".PROCESS) AND ("BUFF".PROCESS <= 35) AND ("IEC_Counter_0_DB".CV = 20);
   IF #_w9 THEN "REVAMP".L30 := "SET VALUE"."PW NO OF PULSES_1"; END_IF;
   #_w10 := #_w9 AND NOT "AUXILIARY".PULSE[20];   // rising edge
   "AUXILIARY".PULSE[20] := #_w9;
   IF #_w10 THEN "TRIGGER" := TRUE; END_IF;
   #_w11 := (1 <= "BUFF".PROCESS) AND ("BUFF".PROCESS <= 35) AND ("IEC_Counter_0_DB".CV = 21);
   IF #_w11 THEN "REVAMP".L30 := "SET VALUE"."WFI DSG TIME"; END_IF;
   #_w12 := #_w11 AND NOT "AUXILIARY".PULSE[21];   // rising edge
   "AUXILIARY".PULSE[21] := #_w11;
   IF #_w12 THEN "TRIGGER" := TRUE; END_IF;
   #_w13 := (1 <= "BUFF".PROCESS) AND ("BUFF".PROCESS <= 35) AND ("IEC_Counter_0_DB".CV = 22);
   IF #_w13 THEN "REVAMP".L30 := "SET VALUE"."WFI WTR TIME"; END_IF;
   #_w14 := #_w13 AND NOT "AUXILIARY".PULSE[22];   // rising edge
   "AUXILIARY".PULSE[22] := #_w13;
   IF #_w14 THEN "TRIGGER" := TRUE; END_IF;
   #_w15 := (1 <= "BUFF".PROCESS) AND ("BUFF".PROCESS <= 35);
   #_w16 := #_w15 AND ("IEC_Counter_0_DB".CV = 23);
   IF #_w16 THEN "REVAMP".L30 := "SET VALUE"."WFI CRC TIME"; END_IF;
   #_w17 := #_w16 AND NOT "AUXILIARY".PULSE[23];   // rising edge
   "AUXILIARY".PULSE[23] := #_w16;
   IF #_w17 THEN "TRIGGER" := TRUE; END_IF;
   #_w18 := #_w15 AND ("IEC_Counter_0_DB".CV = 24);
   IF #_w18 THEN "REVAMP".L30 := "SET VALUE"."WFI DRAIN TIME"; END_IF;
   #_w19 := #_w18 AND NOT "PULSE2";   // rising edge
   "PULSE2" := #_w18;
   IF #_w19 THEN "TRIGGER" := TRUE; END_IF;
   #_w20 := #_w15 AND ("IEC_Counter_0_DB".CV = 25);
   IF #_w20 THEN "REVAMP".L30 := "SET VALUE"."SET WFI COUNTS"; END_IF;
   #_w21 := #_w20 AND NOT "PULSE13";   // rising edge
   "PULSE13" := #_w20;
   IF #_w21 THEN "TRIGGER" := TRUE; END_IF;
   #_w22 := (1 <= "BUFF".PROCESS) AND ("BUFF".PROCESS <= 35) AND ("IEC_Counter_0_DB".CV = 26);
   IF #_w22 THEN "REVAMP".L30 := "SET VALUE"."STERILE TEMP1"; END_IF;
   #_w23 := #_w22 AND NOT "AUXILIARY".PULSE[24];   // rising edge
   "AUXILIARY".PULSE[24] := #_w22;
   IF #_w23 THEN "TRIGGER" := TRUE; END_IF;
   #_w24 := (1 <= "BUFF".PROCESS) AND ("BUFF".PROCESS <= 35) AND ("IEC_Counter_0_DB".CV = 27);
   IF #_w24 THEN "REVAMP".L30 := "SET VALUE"."STERILE HOLD1"; END_IF;
   #_w25 := #_w24 AND NOT "PULSE1";   // rising edge
   "PULSE1" := #_w24;
   IF #_w25 THEN "TRIGGER" := TRUE; END_IF;
   #_w26 := (1 <= "BUFF".PROCESS) AND ("BUFF".PROCESS <= 35) AND ("IEC_Counter_0_DB".CV = 28);
   IF #_w26 THEN "REVAMP".L30 := "SET VALUE"."STERILE TEMP2"; END_IF;
   #_w27 := #_w26 AND NOT "AUXILIARY".PULSE[25];   // rising edge
   "AUXILIARY".PULSE[25] := #_w26;
   IF #_w27 THEN "TRIGGER" := TRUE; END_IF;
   #_w28 := (1 <= "BUFF".PROCESS) AND ("BUFF".PROCESS <= 35) AND ("IEC_Counter_0_DB".CV = 29);
   IF #_w28 THEN "REVAMP".L30 := "SET VALUE"."STERILE HOLD2"; END_IF;
   #_w29 := #_w28 AND NOT "AUXILIARY".PULSE[26];   // rising edge
   "AUXILIARY".PULSE[26] := #_w28;
   IF #_w29 THEN "TRIGGER" := TRUE; END_IF;
   #_w30 := (1 <= "BUFF".PROCESS) AND ("BUFF".PROCESS <= 35) AND ("IEC_Counter_0_DB".CV = 30);
   IF #_w30 THEN "REVAMP".L30 := "SET VALUE"."STERILE TEMP3"; END_IF;
   #_w31 := #_w30 AND NOT "AUXILIARY".PULSE[27];   // rising edge
   "AUXILIARY".PULSE[27] := #_w30;
   IF #_w31 THEN "TRIGGER" := TRUE; END_IF;
   #_w32 := (1 <= "BUFF".PROCESS) AND ("BUFF".PROCESS <= 35) AND ("IEC_Counter_0_DB".CV = 31);
   IF #_w32 THEN "REVAMP".L30 := "SET VALUE"."STERILE HOLD3"; END_IF;
   #_w33 := #_w32 AND NOT "AUXILIARY".PULSE[28];   // rising edge
   "AUXILIARY".PULSE[28] := #_w32;
   IF #_w33 THEN "TRIGGER" := TRUE; END_IF;
   #_w34 := (1 <= "BUFF".PROCESS) AND ("BUFF".PROCESS <= 35) AND ("IEC_Counter_0_DB".CV = 32);
   IF #_w34 THEN "REVAMP".L30 := "SET VALUE"."STERILE TEMP4"; END_IF;
   #_w35 := #_w34 AND NOT "AUXILIARY".PULSE[29];   // rising edge
   "AUXILIARY".PULSE[29] := #_w34;
   IF #_w35 THEN "TRIGGER" := TRUE; END_IF;
   #_w36 := (1 <= "BUFF".PROCESS) AND ("BUFF".PROCESS <= 35) AND ("IEC_Counter_0_DB".CV = 33);
   IF #_w36 THEN "REVAMP".L30 := "SET VALUE"."STERILE HOLD4"; END_IF;
   #_w37 := #_w36 AND NOT "AUXILIARY".PULSE[30];   // rising edge
   "AUXILIARY".PULSE[30] := #_w36;
   IF #_w37 THEN "TRIGGER" := TRUE; END_IF;
   #_w38 := (1 <= "BUFF".PROCESS) AND ("BUFF".PROCESS <= 35);
   #_w39 := #_w38 AND ("IEC_Counter_0_DB".CV = 38);
   IF #_w39 THEN "REVAMP".L30 := "SET VALUE"."OVERSHOOT TEMP"; END_IF;
   #_w40 := #_w39 AND NOT "pulse3";   // rising edge
   "pulse3" := #_w39;
   IF #_w40 THEN "TRIGGER" := TRUE; END_IF;
   #_w41 := #_w38 AND ("IEC_Counter_0_DB".CV = 39);
   IF #_w41 THEN "REVAMP".L30 := "SET VALUE"."ABORT TEMP"; END_IF;
   #_w42 := #_w41 AND NOT "pulse14";   // rising edge
   "pulse14" := #_w41;
   IF #_w42 THEN "TRIGGER" := TRUE; END_IF;
   #_w43 := #_w38 AND ("IEC_Counter_0_DB".CV = 40);
   IF #_w43 THEN "REVAMP".L30 := "SET VALUE"."ABORT DELAY"; END_IF;
   #_w44 := #_w43 AND NOT "pulse15";   // rising edge
   "pulse15" := #_w43;
   IF #_w44 THEN "TRIGGER" := TRUE; END_IF;
   #_w45 := (1 <= "BUFF".PROCESS) AND ("BUFF".PROCESS <= 35) AND ("IEC_Counter_0_DB".CV = 34);
   IF #_w45 THEN "REVAMP".L30 := "SET VALUE"."STERILE EXH PRESS"; END_IF;
   #_w46 := #_w45 AND NOT "AUXILIARY".PULSE[31];   // rising edge
   "AUXILIARY".PULSE[31] := #_w45;
   IF #_w46 THEN "TRIGGER" := TRUE; END_IF;
   #_w47 := (1 <= "BUFF".PROCESS) AND ("BUFF".PROCESS <= 35) AND ("IEC_Counter_0_DB".CV = 35);
   IF #_w47 THEN "REVAMP".L30 := "SET VALUE"."DRY VCC"; END_IF;
   #_w48 := #_w47 AND NOT "AUXILIARY".pulse2[30];   // rising edge
   "AUXILIARY".pulse2[30] := #_w47;
   IF #_w48 THEN "TRIGGER" := TRUE; END_IF;
   #_w49 := (1 <= "BUFF".PROCESS) AND ("BUFF".PROCESS <= 35) AND ("IEC_Counter_0_DB".CV = 36);
   IF #_w49 THEN "REVAMP".L30 := "SET VALUE"."DRY TIME"; END_IF;
   #_w50 := #_w49 AND NOT "AUXILIARY".pulse2[31];   // rising edge
   "AUXILIARY".pulse2[31] := #_w49;
   IF #_w50 THEN "TRIGGER" := TRUE; END_IF;
   #_w51 := (1 <= "BUFF".PROCESS) AND ("BUFF".PROCESS <= 35) AND ("IEC_Counter_0_DB".CV = 37);
   IF #_w51 THEN "REVAMP".L30 := "SET VALUE"."DRY ATS PRESSURE"; END_IF;
   #_w52 := #_w51 AND NOT "AUXILIARY".PULSE[32];   // rising edge
   "AUXILIARY".PULSE[32] := #_w51;
   IF #_w52 THEN "TRIGGER" := TRUE; END_IF;
   #_w53 := NOT "AlwaysTRUE" AND (1 <= "BUFF".PROCESS) AND ("BUFF".PROCESS <= 35) AND ("IEC_Counter_0_DB".CV = 36);
   IF #_w53 THEN "REVAMP".L30 := "SET VALUE"."DRY TIME"; END_IF;
   #_w54 := #_w53 AND NOT "AUXILIARY".PULSE[33];   // rising edge
   "AUXILIARY".PULSE[33] := #_w53;
   IF #_w54 THEN "TRIGGER" := TRUE; END_IF;
END_REGION

REGION Network 8
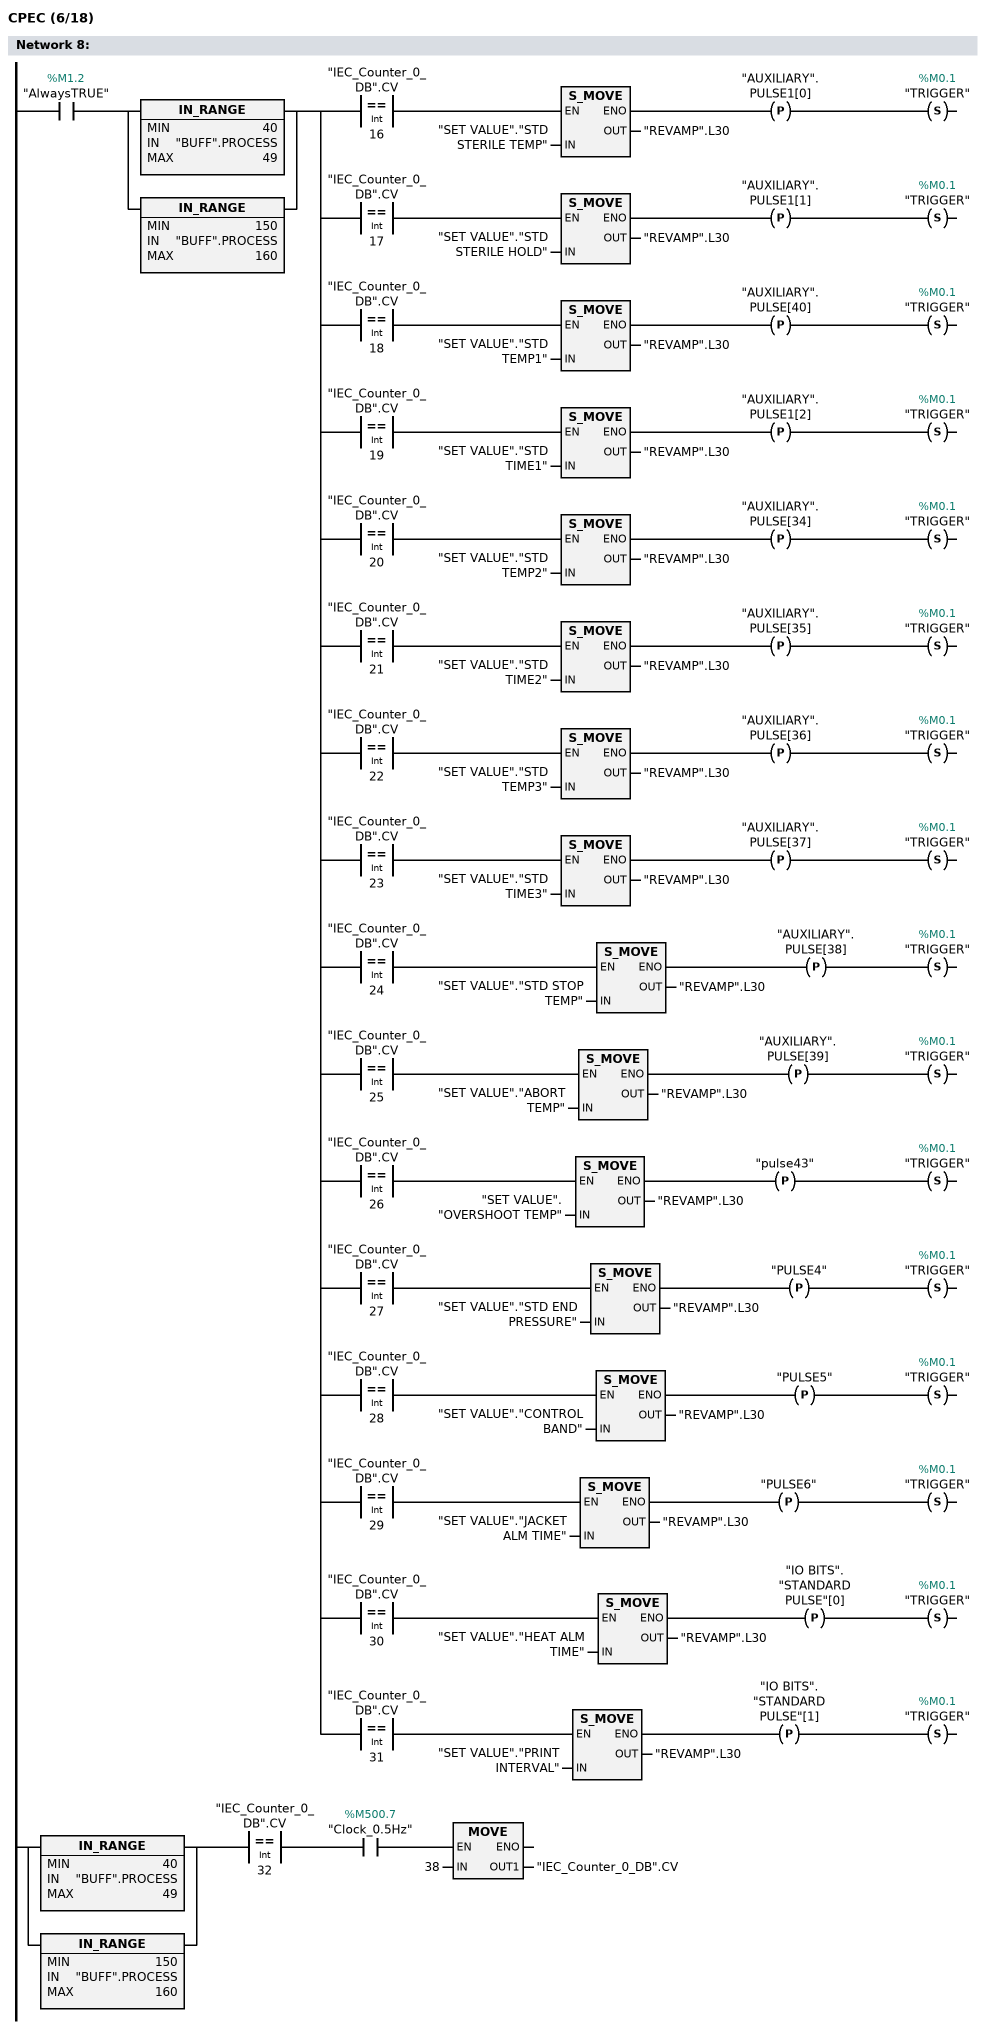
   RUNG wire#powerrail
      Contact( "AlwaysTRUE" )
      wire#w1
      { S7_Templates := "SrcType := Int" } InRange(min := 40, in := "BUFF".PROCESS, max := 49)
      wire#w2
      { S7_Templates := "SrcType := Int" } EQ_Contact(in1 := "IEC_Counter_0_DB".CV, in2 := 16)
      S_Move(in := "SET VALUE"."STD STERILE TEMP", out => "REVAMP".L30)
      P_Trig( "AUXILIARY".PULSE1[0] )
      S_Coil( "TRIGGER" )
   END_RUNG
   RUNG wire#w1
      { S7_Templates := "SrcType := Int" } InRange(min := 150, in := "BUFF".PROCESS, max := 160)
   END_RUNG wire#w2
   RUNG wire#w2
      { S7_Templates := "SrcType := Int" } EQ_Contact(in1 := "IEC_Counter_0_DB".CV, in2 := 17)
      S_Move(in := "SET VALUE"."STD STERILE HOLD", out => "REVAMP".L30)
      P_Trig( "AUXILIARY".PULSE1[1] )
      S_Coil( "TRIGGER" )
   END_RUNG
   RUNG wire#w2
      { S7_Templates := "SrcType := Int" } EQ_Contact(in1 := "IEC_Counter_0_DB".CV, in2 := 18)
      S_Move(in := "SET VALUE"."STD TEMP1", out => "REVAMP".L30)
      P_Trig( "AUXILIARY".PULSE[40] )
      S_Coil( "TRIGGER" )
   END_RUNG
   RUNG wire#w2
      { S7_Templates := "SrcType := Int" } EQ_Contact(in1 := "IEC_Counter_0_DB".CV, in2 := 19)
      S_Move(in := "SET VALUE"."STD TIME1", out => "REVAMP".L30)
      P_Trig( "AUXILIARY".PULSE1[2] )
      S_Coil( "TRIGGER" )
   END_RUNG
   RUNG wire#w2
      { S7_Templates := "SrcType := Int" } EQ_Contact(in1 := "IEC_Counter_0_DB".CV, in2 := 20)
      S_Move(in := "SET VALUE"."STD TEMP2", out => "REVAMP".L30)
      P_Trig( "AUXILIARY".PULSE[34] )
      S_Coil( "TRIGGER" )
   END_RUNG
   RUNG wire#w2
      { S7_Templates := "SrcType := Int" } EQ_Contact(in1 := "IEC_Counter_0_DB".CV, in2 := 21)
      S_Move(in := "SET VALUE"."STD TIME2", out => "REVAMP".L30)
      P_Trig( "AUXILIARY".PULSE[35] )
      S_Coil( "TRIGGER" )
   END_RUNG
   RUNG wire#w2
      { S7_Templates := "SrcType := Int" } EQ_Contact(in1 := "IEC_Counter_0_DB".CV, in2 := 22)
      S_Move(in := "SET VALUE"."STD TEMP3", out => "REVAMP".L30)
      P_Trig( "AUXILIARY".PULSE[36] )
      S_Coil( "TRIGGER" )
   END_RUNG
   RUNG wire#w2
      { S7_Templates := "SrcType := Int" } EQ_Contact(in1 := "IEC_Counter_0_DB".CV, in2 := 23)
      S_Move(in := "SET VALUE"."STD TIME3", out => "REVAMP".L30)
      P_Trig( "AUXILIARY".PULSE[37] )
      S_Coil( "TRIGGER" )
   END_RUNG
   RUNG wire#w2
      { S7_Templates := "SrcType := Int" } EQ_Contact(in1 := "IEC_Counter_0_DB".CV, in2 := 24)
      S_Move(in := "SET VALUE"."STD STOP TEMP", out => "REVAMP".L30)
      P_Trig( "AUXILIARY".PULSE[38] )
      S_Coil( "TRIGGER" )
   END_RUNG
   RUNG wire#w2
      { S7_Templates := "SrcType := Int" } EQ_Contact(in1 := "IEC_Counter_0_DB".CV, in2 := 25)
      S_Move(in := "SET VALUE"."ABORT TEMP", out => "REVAMP".L30)
      P_Trig( "AUXILIARY".PULSE[39] )
      S_Coil( "TRIGGER" )
   END_RUNG
   RUNG wire#w2
      { S7_Templates := "SrcType := Int" } EQ_Contact(in1 := "IEC_Counter_0_DB".CV, in2 := 26)
      S_Move(in := "SET VALUE"."OVERSHOOT TEMP", out => "REVAMP".L30)
      P_Trig( "pulse43" )
      S_Coil( "TRIGGER" )
   END_RUNG
   RUNG wire#w2
      { S7_Templates := "SrcType := Int" } EQ_Contact(in1 := "IEC_Counter_0_DB".CV, in2 := 27)
      S_Move(in := "SET VALUE"."STD END PRESSURE", out => "REVAMP".L30)
      P_Trig( "PULSE4" )
      S_Coil( "TRIGGER" )
   END_RUNG
   RUNG wire#w2
      { S7_Templates := "SrcType := Int" } EQ_Contact(in1 := "IEC_Counter_0_DB".CV, in2 := 28)
      S_Move(in := "SET VALUE"."CONTROL BAND", out => "REVAMP".L30)
      P_Trig( "PULSE5" )
      S_Coil( "TRIGGER" )
   END_RUNG
   RUNG wire#w2
      { S7_Templates := "SrcType := Int" } EQ_Contact(in1 := "IEC_Counter_0_DB".CV, in2 := 29)
      S_Move(in := "SET VALUE"."JACKET ALM TIME", out => "REVAMP".L30)
      P_Trig( "PULSE6" )
      S_Coil( "TRIGGER" )
   END_RUNG
   RUNG wire#w2
      { S7_Templates := "SrcType := Int" } EQ_Contact(in1 := "IEC_Counter_0_DB".CV, in2 := 30)
      S_Move(in := "SET VALUE"."HEAT ALM TIME", out => "REVAMP".L30)
      P_Trig( "IO BITS"."STANDARD PULSE"[0] )
      S_Coil( "TRIGGER" )
   END_RUNG
   RUNG wire#w2
      { S7_Templates := "SrcType := Int" } EQ_Contact(in1 := "IEC_Counter_0_DB".CV, in2 := 31)
      S_Move(in := "SET VALUE"."PRINT INTERVAL", out => "REVAMP".L30)
      P_Trig( "IO BITS"."STANDARD PULSE"[1] )
      S_Coil( "TRIGGER" )
   END_RUNG
   RUNG wire#powerrail
      { S7_Templates := "SrcType := Int" } InRange(min := 40, in := "BUFF".PROCESS, max := 49)
      wire#w3
      { S7_Templates := "SrcType := Int" } EQ_Contact(in1 := "IEC_Counter_0_DB".CV, in2 := 32)
      Contact( "Clock_0.5Hz" )
      Move(in := 38, out1 => "IEC_Counter_0_DB".CV)
   END_RUNG
   RUNG wire#powerrail
      { S7_Templates := "SrcType := Int" } InRange(min := 150, in := "BUFF".PROCESS, max := 160)
   END_RUNG wire#w3
   // the same network as SCL:
   #_w1 := "AlwaysTRUE" AND (((40 <= "BUFF".PROCESS) AND ("BUFF".PROCESS <= 49)) OR ((150 <= "BUFF".PROCESS) AND ("BUFF".PROCESS <= 160)));
   #_w2 := #_w1 AND ("IEC_Counter_0_DB".CV = 16);
   IF #_w2 THEN "REVAMP".L30 := "SET VALUE"."STD STERILE TEMP"; END_IF;
   #_w3 := #_w2 AND NOT "AUXILIARY".PULSE1[0];   // rising edge
   "AUXILIARY".PULSE1[0] := #_w2;
   IF #_w3 THEN "TRIGGER" := TRUE; END_IF;
   #_w4 := #_w1 AND ("IEC_Counter_0_DB".CV = 17);
   IF #_w4 THEN "REVAMP".L30 := "SET VALUE"."STD STERILE HOLD"; END_IF;
   #_w5 := #_w4 AND NOT "AUXILIARY".PULSE1[1];   // rising edge
   "AUXILIARY".PULSE1[1] := #_w4;
   IF #_w5 THEN "TRIGGER" := TRUE; END_IF;
   #_w6 := #_w1 AND ("IEC_Counter_0_DB".CV = 18);
   IF #_w6 THEN "REVAMP".L30 := "SET VALUE"."STD TEMP1"; END_IF;
   #_w7 := #_w6 AND NOT "AUXILIARY".PULSE[40];   // rising edge
   "AUXILIARY".PULSE[40] := #_w6;
   IF #_w7 THEN "TRIGGER" := TRUE; END_IF;
   #_w8 := #_w1 AND ("IEC_Counter_0_DB".CV = 19);
   IF #_w8 THEN "REVAMP".L30 := "SET VALUE"."STD TIME1"; END_IF;
   #_w9 := #_w8 AND NOT "AUXILIARY".PULSE1[2];   // rising edge
   "AUXILIARY".PULSE1[2] := #_w8;
   IF #_w9 THEN "TRIGGER" := TRUE; END_IF;
   #_w10 := #_w1 AND ("IEC_Counter_0_DB".CV = 20);
   IF #_w10 THEN "REVAMP".L30 := "SET VALUE"."STD TEMP2"; END_IF;
   #_w11 := #_w10 AND NOT "AUXILIARY".PULSE[34];   // rising edge
   "AUXILIARY".PULSE[34] := #_w10;
   IF #_w11 THEN "TRIGGER" := TRUE; END_IF;
   #_w12 := #_w1 AND ("IEC_Counter_0_DB".CV = 21);
   IF #_w12 THEN "REVAMP".L30 := "SET VALUE"."STD TIME2"; END_IF;
   #_w13 := #_w12 AND NOT "AUXILIARY".PULSE[35];   // rising edge
   "AUXILIARY".PULSE[35] := #_w12;
   IF #_w13 THEN "TRIGGER" := TRUE; END_IF;
   #_w14 := #_w1 AND ("IEC_Counter_0_DB".CV = 22);
   IF #_w14 THEN "REVAMP".L30 := "SET VALUE"."STD TEMP3"; END_IF;
   #_w15 := #_w14 AND NOT "AUXILIARY".PULSE[36];   // rising edge
   "AUXILIARY".PULSE[36] := #_w14;
   IF #_w15 THEN "TRIGGER" := TRUE; END_IF;
   #_w16 := #_w1 AND ("IEC_Counter_0_DB".CV = 23);
   IF #_w16 THEN "REVAMP".L30 := "SET VALUE"."STD TIME3"; END_IF;
   #_w17 := #_w16 AND NOT "AUXILIARY".PULSE[37];   // rising edge
   "AUXILIARY".PULSE[37] := #_w16;
   IF #_w17 THEN "TRIGGER" := TRUE; END_IF;
   #_w18 := #_w1 AND ("IEC_Counter_0_DB".CV = 24);
   IF #_w18 THEN "REVAMP".L30 := "SET VALUE"."STD STOP TEMP"; END_IF;
   #_w19 := #_w18 AND NOT "AUXILIARY".PULSE[38];   // rising edge
   "AUXILIARY".PULSE[38] := #_w18;
   IF #_w19 THEN "TRIGGER" := TRUE; END_IF;
   #_w20 := #_w1 AND ("IEC_Counter_0_DB".CV = 25);
   IF #_w20 THEN "REVAMP".L30 := "SET VALUE"."ABORT TEMP"; END_IF;
   #_w21 := #_w20 AND NOT "AUXILIARY".PULSE[39];   // rising edge
   "AUXILIARY".PULSE[39] := #_w20;
   IF #_w21 THEN "TRIGGER" := TRUE; END_IF;
   #_w22 := #_w1 AND ("IEC_Counter_0_DB".CV = 26);
   IF #_w22 THEN "REVAMP".L30 := "SET VALUE"."OVERSHOOT TEMP"; END_IF;
   #_w23 := #_w22 AND NOT "pulse43";   // rising edge
   "pulse43" := #_w22;
   IF #_w23 THEN "TRIGGER" := TRUE; END_IF;
   #_w24 := #_w1 AND ("IEC_Counter_0_DB".CV = 27);
   IF #_w24 THEN "REVAMP".L30 := "SET VALUE"."STD END PRESSURE"; END_IF;
   #_w25 := #_w24 AND NOT "PULSE4";   // rising edge
   "PULSE4" := #_w24;
   IF #_w25 THEN "TRIGGER" := TRUE; END_IF;
   #_w26 := #_w1 AND ("IEC_Counter_0_DB".CV = 28);
   IF #_w26 THEN "REVAMP".L30 := "SET VALUE"."CONTROL BAND"; END_IF;
   #_w27 := #_w26 AND NOT "PULSE5";   // rising edge
   "PULSE5" := #_w26;
   IF #_w27 THEN "TRIGGER" := TRUE; END_IF;
   #_w28 := #_w1 AND ("IEC_Counter_0_DB".CV = 29);
   IF #_w28 THEN "REVAMP".L30 := "SET VALUE"."JACKET ALM TIME"; END_IF;
   #_w29 := #_w28 AND NOT "PULSE6";   // rising edge
   "PULSE6" := #_w28;
   IF #_w29 THEN "TRIGGER" := TRUE; END_IF;
   #_w30 := #_w1 AND ("IEC_Counter_0_DB".CV = 30);
   IF #_w30 THEN "REVAMP".L30 := "SET VALUE"."HEAT ALM TIME"; END_IF;
   #_w31 := #_w30 AND NOT "IO BITS"."STANDARD PULSE"[0];   // rising edge
   "IO BITS"."STANDARD PULSE"[0] := #_w30;
   IF #_w31 THEN "TRIGGER" := TRUE; END_IF;
   #_w32 := #_w1 AND ("IEC_Counter_0_DB".CV = 31);
   IF #_w32 THEN "REVAMP".L30 := "SET VALUE"."PRINT INTERVAL"; END_IF;
   #_w33 := #_w32 AND NOT "IO BITS"."STANDARD PULSE"[1];   // rising edge
   "IO BITS"."STANDARD PULSE"[1] := #_w32;
   IF #_w33 THEN "TRIGGER" := TRUE; END_IF;
   IF (((40 <= "BUFF".PROCESS) AND ("BUFF".PROCESS <= 49)) OR ((150 <= "BUFF".PROCESS) AND ("BUFF".PROCESS <= 160))) AND ("IEC_Counter_0_DB".CV = 32) AND "Clock_0.5Hz" THEN
       "IEC_Counter_0_DB".CV := 38;
   END_IF;
END_REGION

REGION Network 9
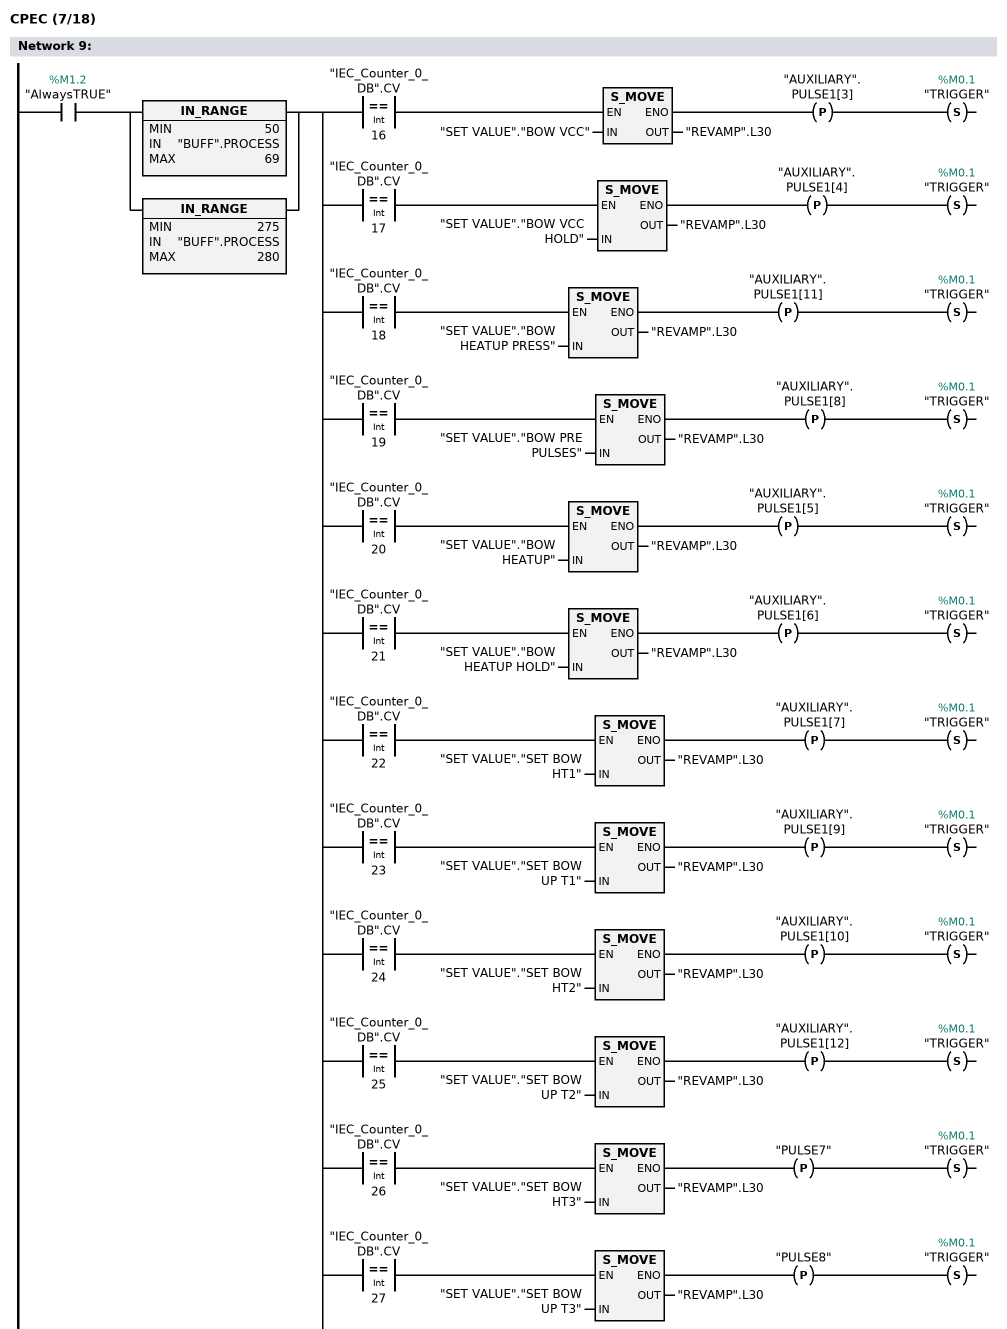
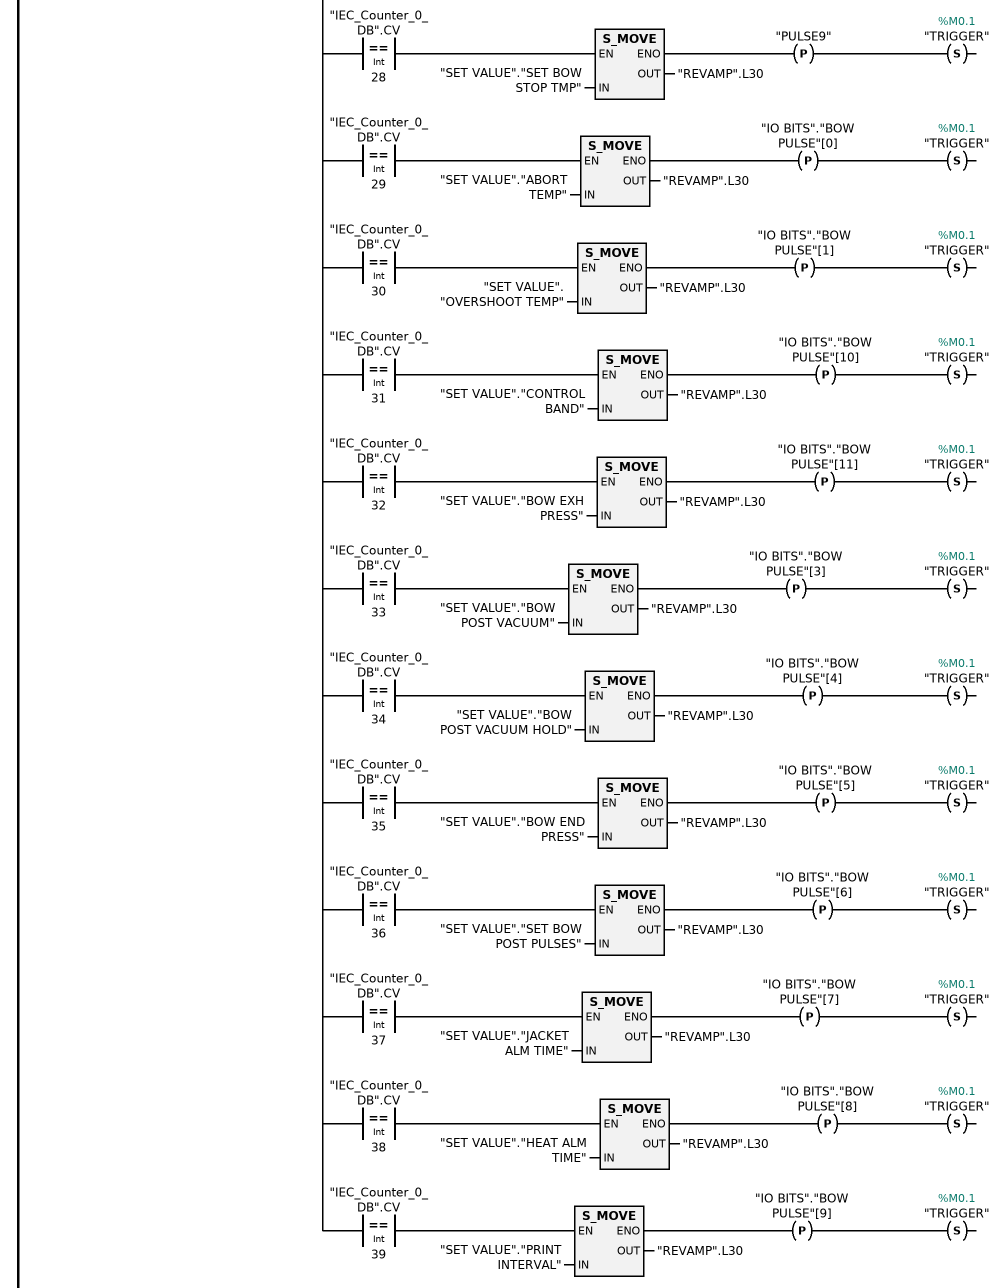
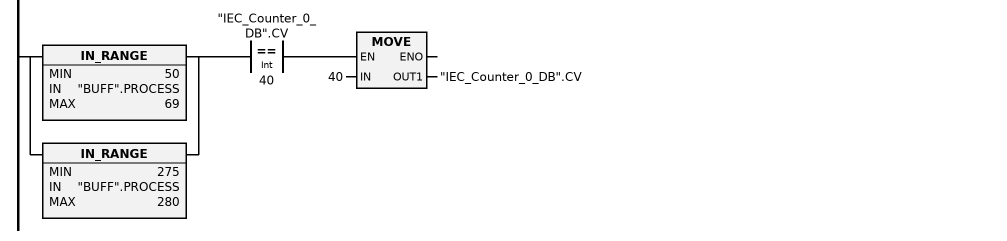
   RUNG wire#powerrail
      Contact( "AlwaysTRUE" )
      wire#w1
      { S7_Templates := "SrcType := Int" } InRange(min := 50, in := "BUFF".PROCESS, max := 69)
      wire#w2
      { S7_Templates := "SrcType := Int" } EQ_Contact(in1 := "IEC_Counter_0_DB".CV, in2 := 16)
      S_Move(in := "SET VALUE"."BOW VCC", out => "REVAMP".L30)
      P_Trig( "AUXILIARY".PULSE1[3] )
      S_Coil( "TRIGGER" )
   END_RUNG
   RUNG wire#w1
      { S7_Templates := "SrcType := Int" } InRange(min := 275, in := "BUFF".PROCESS, max := 280)
   END_RUNG wire#w2
   RUNG wire#w2
      { S7_Templates := "SrcType := Int" } EQ_Contact(in1 := "IEC_Counter_0_DB".CV, in2 := 17)
      S_Move(in := "SET VALUE"."BOW VCC HOLD", out => "REVAMP".L30)
      P_Trig( "AUXILIARY".PULSE1[4] )
      S_Coil( "TRIGGER" )
   END_RUNG
   RUNG wire#w2
      { S7_Templates := "SrcType := Int" } EQ_Contact(in1 := "IEC_Counter_0_DB".CV, in2 := 18)
      S_Move(in := "SET VALUE"."BOW HEATUP PRESS", out => "REVAMP".L30)
      P_Trig( "AUXILIARY".PULSE1[11] )
      S_Coil( "TRIGGER" )
   END_RUNG
   RUNG wire#w2
      { S7_Templates := "SrcType := Int" } EQ_Contact(in1 := "IEC_Counter_0_DB".CV, in2 := 19)
      S_Move(in := "SET VALUE"."BOW PRE PULSES", out => "REVAMP".L30)
      P_Trig( "AUXILIARY".PULSE1[8] )
      S_Coil( "TRIGGER" )
   END_RUNG
   RUNG wire#w2
      { S7_Templates := "SrcType := Int" } EQ_Contact(in1 := "IEC_Counter_0_DB".CV, in2 := 20)
      S_Move(in := "SET VALUE"."BOW HEATUP", out => "REVAMP".L30)
      P_Trig( "AUXILIARY".PULSE1[5] )
      S_Coil( "TRIGGER" )
   END_RUNG
   RUNG wire#w2
      { S7_Templates := "SrcType := Int" } EQ_Contact(in1 := "IEC_Counter_0_DB".CV, in2 := 21)
      S_Move(in := "SET VALUE"."BOW HEATUP HOLD", out => "REVAMP".L30)
      P_Trig( "AUXILIARY".PULSE1[6] )
      S_Coil( "TRIGGER" )
   END_RUNG
   RUNG wire#w2
      { S7_Templates := "SrcType := Int" } EQ_Contact(in1 := "IEC_Counter_0_DB".CV, in2 := 22)
      S_Move(in := "SET VALUE"."SET BOW HT1", out => "REVAMP".L30)
      P_Trig( "AUXILIARY".PULSE1[7] )
      S_Coil( "TRIGGER" )
   END_RUNG
   RUNG wire#w2
      { S7_Templates := "SrcType := Int" } EQ_Contact(in1 := "IEC_Counter_0_DB".CV, in2 := 23)
      S_Move(in := "SET VALUE"."SET BOW UP T1", out => "REVAMP".L30)
      P_Trig( "AUXILIARY".PULSE1[9] )
      S_Coil( "TRIGGER" )
   END_RUNG
   RUNG wire#w2
      { S7_Templates := "SrcType := Int" } EQ_Contact(in1 := "IEC_Counter_0_DB".CV, in2 := 24)
      S_Move(in := "SET VALUE"."SET BOW HT2", out => "REVAMP".L30)
      P_Trig( "AUXILIARY".PULSE1[10] )
      S_Coil( "TRIGGER" )
   END_RUNG
   RUNG wire#w2
      { S7_Templates := "SrcType := Int" } EQ_Contact(in1 := "IEC_Counter_0_DB".CV, in2 := 25)
      S_Move(in := "SET VALUE"."SET BOW UP T2", out => "REVAMP".L30)
      P_Trig( "AUXILIARY".PULSE1[12] )
      S_Coil( "TRIGGER" )
   END_RUNG
   RUNG wire#w2
      { S7_Templates := "SrcType := Int" } EQ_Contact(in1 := "IEC_Counter_0_DB".CV, in2 := 26)
      S_Move(in := "SET VALUE"."SET BOW HT3", out => "REVAMP".L30)
      P_Trig( "PULSE7" )
      S_Coil( "TRIGGER" )
   END_RUNG
   RUNG wire#w2
      { S7_Templates := "SrcType := Int" } EQ_Contact(in1 := "IEC_Counter_0_DB".CV, in2 := 27)
      S_Move(in := "SET VALUE"."SET BOW UP T3", out => "REVAMP".L30)
      P_Trig( "PULSE8" )
      S_Coil( "TRIGGER" )
   END_RUNG
   RUNG wire#w2
      { S7_Templates := "SrcType := Int" } EQ_Contact(in1 := "IEC_Counter_0_DB".CV, in2 := 28)
      S_Move(in := "SET VALUE"."SET BOW STOP TMP", out => "REVAMP".L30)
      P_Trig( "PULSE9" )
      S_Coil( "TRIGGER" )
   END_RUNG
   RUNG wire#w2
      { S7_Templates := "SrcType := Int" } EQ_Contact(in1 := "IEC_Counter_0_DB".CV, in2 := 29)
      S_Move(in := "SET VALUE"."ABORT TEMP", out => "REVAMP".L30)
      P_Trig( "IO BITS"."BOW PULSE"[0] )
      S_Coil( "TRIGGER" )
   END_RUNG
   RUNG wire#w2
      { S7_Templates := "SrcType := Int" } EQ_Contact(in1 := "IEC_Counter_0_DB".CV, in2 := 30)
      S_Move(in := "SET VALUE"."OVERSHOOT TEMP", out => "REVAMP".L30)
      P_Trig( "IO BITS"."BOW PULSE"[1] )
      S_Coil( "TRIGGER" )
   END_RUNG
   RUNG wire#w2
      { S7_Templates := "SrcType := Int" } EQ_Contact(in1 := "IEC_Counter_0_DB".CV, in2 := 31)
      S_Move(in := "SET VALUE"."CONTROL BAND", out => "REVAMP".L30)
      P_Trig( "IO BITS"."BOW PULSE"[10] )
      S_Coil( "TRIGGER" )
   END_RUNG
   RUNG wire#w2
      { S7_Templates := "SrcType := Int" } EQ_Contact(in1 := "IEC_Counter_0_DB".CV, in2 := 32)
      S_Move(in := "SET VALUE"."BOW EXH PRESS", out => "REVAMP".L30)
      P_Trig( "IO BITS"."BOW PULSE"[11] )
      S_Coil( "TRIGGER" )
   END_RUNG
   RUNG wire#w2
      { S7_Templates := "SrcType := Int" } EQ_Contact(in1 := "IEC_Counter_0_DB".CV, in2 := 33)
      S_Move(in := "SET VALUE"."BOW POST VACUUM", out => "REVAMP".L30)
      P_Trig( "IO BITS"."BOW PULSE"[3] )
      S_Coil( "TRIGGER" )
   END_RUNG
   RUNG wire#w2
      { S7_Templates := "SrcType := Int" } EQ_Contact(in1 := "IEC_Counter_0_DB".CV, in2 := 34)
      S_Move(in := "SET VALUE"."BOW POST VACUUM HOLD", out => "REVAMP".L30)
      P_Trig( "IO BITS"."BOW PULSE"[4] )
      S_Coil( "TRIGGER" )
   END_RUNG
   RUNG wire#w2
      { S7_Templates := "SrcType := Int" } EQ_Contact(in1 := "IEC_Counter_0_DB".CV, in2 := 35)
      S_Move(in := "SET VALUE"."BOW END PRESS", out => "REVAMP".L30)
      P_Trig( "IO BITS"."BOW PULSE"[5] )
      S_Coil( "TRIGGER" )
   END_RUNG
   RUNG wire#w2
      { S7_Templates := "SrcType := Int" } EQ_Contact(in1 := "IEC_Counter_0_DB".CV, in2 := 36)
      S_Move(in := "SET VALUE"."SET BOW POST PULSES", out => "REVAMP".L30)
      P_Trig( "IO BITS"."BOW PULSE"[6] )
      S_Coil( "TRIGGER" )
   END_RUNG
   RUNG wire#w2
      { S7_Templates := "SrcType := Int" } EQ_Contact(in1 := "IEC_Counter_0_DB".CV, in2 := 37)
      S_Move(in := "SET VALUE"."JACKET ALM TIME", out => "REVAMP".L30)
      P_Trig( "IO BITS"."BOW PULSE"[7] )
      S_Coil( "TRIGGER" )
   END_RUNG
   RUNG wire#w2
      { S7_Templates := "SrcType := Int" } EQ_Contact(in1 := "IEC_Counter_0_DB".CV, in2 := 38)
      S_Move(in := "SET VALUE"."HEAT ALM TIME", out => "REVAMP".L30)
      P_Trig( "IO BITS"."BOW PULSE"[8] )
      S_Coil( "TRIGGER" )
   END_RUNG
   RUNG wire#w2
      { S7_Templates := "SrcType := Int" } EQ_Contact(in1 := "IEC_Counter_0_DB".CV, in2 := 39)
      S_Move(in := "SET VALUE"."PRINT INTERVAL", out => "REVAMP".L30)
      P_Trig( "IO BITS"."BOW PULSE"[9] )
      S_Coil( "TRIGGER" )
   END_RUNG
   RUNG wire#powerrail
      { S7_Templates := "SrcType := Int" } InRange(min := 50, in := "BUFF".PROCESS, max := 69)
      wire#w3
      { S7_Templates := "SrcType := Int" } EQ_Contact(in1 := "IEC_Counter_0_DB".CV, in2 := 40)
      Move(in := 40, out1 => "IEC_Counter_0_DB".CV)
   END_RUNG
   RUNG wire#powerrail
      { S7_Templates := "SrcType := Int" } InRange(min := 275, in := "BUFF".PROCESS, max := 280)
   END_RUNG wire#w3
   // the same network as SCL:
   #_w1 := "AlwaysTRUE" AND (((50 <= "BUFF".PROCESS) AND ("BUFF".PROCESS <= 69)) OR ((275 <= "BUFF".PROCESS) AND ("BUFF".PROCESS <= 280)));
   #_w2 := #_w1 AND ("IEC_Counter_0_DB".CV = 16);
   IF #_w2 THEN "REVAMP".L30 := "SET VALUE"."BOW VCC"; END_IF;
   #_w3 := #_w2 AND NOT "AUXILIARY".PULSE1[3];   // rising edge
   "AUXILIARY".PULSE1[3] := #_w2;
   IF #_w3 THEN "TRIGGER" := TRUE; END_IF;
   #_w4 := #_w1 AND ("IEC_Counter_0_DB".CV = 17);
   IF #_w4 THEN "REVAMP".L30 := "SET VALUE"."BOW VCC HOLD"; END_IF;
   #_w5 := #_w4 AND NOT "AUXILIARY".PULSE1[4];   // rising edge
   "AUXILIARY".PULSE1[4] := #_w4;
   IF #_w5 THEN "TRIGGER" := TRUE; END_IF;
   #_w6 := #_w1 AND ("IEC_Counter_0_DB".CV = 18);
   IF #_w6 THEN "REVAMP".L30 := "SET VALUE"."BOW HEATUP PRESS"; END_IF;
   #_w7 := #_w6 AND NOT "AUXILIARY".PULSE1[11];   // rising edge
   "AUXILIARY".PULSE1[11] := #_w6;
   IF #_w7 THEN "TRIGGER" := TRUE; END_IF;
   #_w8 := #_w1 AND ("IEC_Counter_0_DB".CV = 19);
   IF #_w8 THEN "REVAMP".L30 := "SET VALUE"."BOW PRE PULSES"; END_IF;
   #_w9 := #_w8 AND NOT "AUXILIARY".PULSE1[8];   // rising edge
   "AUXILIARY".PULSE1[8] := #_w8;
   IF #_w9 THEN "TRIGGER" := TRUE; END_IF;
   #_w10 := #_w1 AND ("IEC_Counter_0_DB".CV = 20);
   IF #_w10 THEN "REVAMP".L30 := "SET VALUE"."BOW HEATUP"; END_IF;
   #_w11 := #_w10 AND NOT "AUXILIARY".PULSE1[5];   // rising edge
   "AUXILIARY".PULSE1[5] := #_w10;
   IF #_w11 THEN "TRIGGER" := TRUE; END_IF;
   #_w12 := #_w1 AND ("IEC_Counter_0_DB".CV = 21);
   IF #_w12 THEN "REVAMP".L30 := "SET VALUE"."BOW HEATUP HOLD"; END_IF;
   #_w13 := #_w12 AND NOT "AUXILIARY".PULSE1[6];   // rising edge
   "AUXILIARY".PULSE1[6] := #_w12;
   IF #_w13 THEN "TRIGGER" := TRUE; END_IF;
   #_w14 := #_w1 AND ("IEC_Counter_0_DB".CV = 22);
   IF #_w14 THEN "REVAMP".L30 := "SET VALUE"."SET BOW HT1"; END_IF;
   #_w15 := #_w14 AND NOT "AUXILIARY".PULSE1[7];   // rising edge
   "AUXILIARY".PULSE1[7] := #_w14;
   IF #_w15 THEN "TRIGGER" := TRUE; END_IF;
   #_w16 := #_w1 AND ("IEC_Counter_0_DB".CV = 23);
   IF #_w16 THEN "REVAMP".L30 := "SET VALUE"."SET BOW UP T1"; END_IF;
   #_w17 := #_w16 AND NOT "AUXILIARY".PULSE1[9];   // rising edge
   "AUXILIARY".PULSE1[9] := #_w16;
   IF #_w17 THEN "TRIGGER" := TRUE; END_IF;
   #_w18 := #_w1 AND ("IEC_Counter_0_DB".CV = 24);
   IF #_w18 THEN "REVAMP".L30 := "SET VALUE"."SET BOW HT2"; END_IF;
   #_w19 := #_w18 AND NOT "AUXILIARY".PULSE1[10];   // rising edge
   "AUXILIARY".PULSE1[10] := #_w18;
   IF #_w19 THEN "TRIGGER" := TRUE; END_IF;
   #_w20 := #_w1 AND ("IEC_Counter_0_DB".CV = 25);
   IF #_w20 THEN "REVAMP".L30 := "SET VALUE"."SET BOW UP T2"; END_IF;
   #_w21 := #_w20 AND NOT "AUXILIARY".PULSE1[12];   // rising edge
   "AUXILIARY".PULSE1[12] := #_w20;
   IF #_w21 THEN "TRIGGER" := TRUE; END_IF;
   #_w22 := #_w1 AND ("IEC_Counter_0_DB".CV = 26);
   IF #_w22 THEN "REVAMP".L30 := "SET VALUE"."SET BOW HT3"; END_IF;
   #_w23 := #_w22 AND NOT "PULSE7";   // rising edge
   "PULSE7" := #_w22;
   IF #_w23 THEN "TRIGGER" := TRUE; END_IF;
   #_w24 := #_w1 AND ("IEC_Counter_0_DB".CV = 27);
   IF #_w24 THEN "REVAMP".L30 := "SET VALUE"."SET BOW UP T3"; END_IF;
   #_w25 := #_w24 AND NOT "PULSE8";   // rising edge
   "PULSE8" := #_w24;
   IF #_w25 THEN "TRIGGER" := TRUE; END_IF;
   #_w26 := #_w1 AND ("IEC_Counter_0_DB".CV = 28);
   IF #_w26 THEN "REVAMP".L30 := "SET VALUE"."SET BOW STOP TMP"; END_IF;
   #_w27 := #_w26 AND NOT "PULSE9";   // rising edge
   "PULSE9" := #_w26;
   IF #_w27 THEN "TRIGGER" := TRUE; END_IF;
   #_w28 := #_w1 AND ("IEC_Counter_0_DB".CV = 29);
   IF #_w28 THEN "REVAMP".L30 := "SET VALUE"."ABORT TEMP"; END_IF;
   #_w29 := #_w28 AND NOT "IO BITS"."BOW PULSE"[0];   // rising edge
   "IO BITS"."BOW PULSE"[0] := #_w28;
   IF #_w29 THEN "TRIGGER" := TRUE; END_IF;
   #_w30 := #_w1 AND ("IEC_Counter_0_DB".CV = 30);
   IF #_w30 THEN "REVAMP".L30 := "SET VALUE"."OVERSHOOT TEMP"; END_IF;
   #_w31 := #_w30 AND NOT "IO BITS"."BOW PULSE"[1];   // rising edge
   "IO BITS"."BOW PULSE"[1] := #_w30;
   IF #_w31 THEN "TRIGGER" := TRUE; END_IF;
   #_w32 := #_w1 AND ("IEC_Counter_0_DB".CV = 31);
   IF #_w32 THEN "REVAMP".L30 := "SET VALUE"."CONTROL BAND"; END_IF;
   #_w33 := #_w32 AND NOT "IO BITS"."BOW PULSE"[10];   // rising edge
   "IO BITS"."BOW PULSE"[10] := #_w32;
   IF #_w33 THEN "TRIGGER" := TRUE; END_IF;
   #_w34 := #_w1 AND ("IEC_Counter_0_DB".CV = 32);
   IF #_w34 THEN "REVAMP".L30 := "SET VALUE"."BOW EXH PRESS"; END_IF;
   #_w35 := #_w34 AND NOT "IO BITS"."BOW PULSE"[11];   // rising edge
   "IO BITS"."BOW PULSE"[11] := #_w34;
   IF #_w35 THEN "TRIGGER" := TRUE; END_IF;
   #_w36 := #_w1 AND ("IEC_Counter_0_DB".CV = 33);
   IF #_w36 THEN "REVAMP".L30 := "SET VALUE"."BOW POST VACUUM"; END_IF;
   #_w37 := #_w36 AND NOT "IO BITS"."BOW PULSE"[3];   // rising edge
   "IO BITS"."BOW PULSE"[3] := #_w36;
   IF #_w37 THEN "TRIGGER" := TRUE; END_IF;
   #_w38 := #_w1 AND ("IEC_Counter_0_DB".CV = 34);
   IF #_w38 THEN "REVAMP".L30 := "SET VALUE"."BOW POST VACUUM HOLD"; END_IF;
   #_w39 := #_w38 AND NOT "IO BITS"."BOW PULSE"[4];   // rising edge
   "IO BITS"."BOW PULSE"[4] := #_w38;
   IF #_w39 THEN "TRIGGER" := TRUE; END_IF;
   #_w40 := #_w1 AND ("IEC_Counter_0_DB".CV = 35);
   IF #_w40 THEN "REVAMP".L30 := "SET VALUE"."BOW END PRESS"; END_IF;
   #_w41 := #_w40 AND NOT "IO BITS"."BOW PULSE"[5];   // rising edge
   "IO BITS"."BOW PULSE"[5] := #_w40;
   IF #_w41 THEN "TRIGGER" := TRUE; END_IF;
   #_w42 := #_w1 AND ("IEC_Counter_0_DB".CV = 36);
   IF #_w42 THEN "REVAMP".L30 := "SET VALUE"."SET BOW POST PULSES"; END_IF;
   #_w43 := #_w42 AND NOT "IO BITS"."BOW PULSE"[6];   // rising edge
   "IO BITS"."BOW PULSE"[6] := #_w42;
   IF #_w43 THEN "TRIGGER" := TRUE; END_IF;
   #_w44 := #_w1 AND ("IEC_Counter_0_DB".CV = 37);
   IF #_w44 THEN "REVAMP".L30 := "SET VALUE"."JACKET ALM TIME"; END_IF;
   #_w45 := #_w44 AND NOT "IO BITS"."BOW PULSE"[7];   // rising edge
   "IO BITS"."BOW PULSE"[7] := #_w44;
   IF #_w45 THEN "TRIGGER" := TRUE; END_IF;
   #_w46 := #_w1 AND ("IEC_Counter_0_DB".CV = 38);
   IF #_w46 THEN "REVAMP".L30 := "SET VALUE"."HEAT ALM TIME"; END_IF;
   #_w47 := #_w46 AND NOT "IO BITS"."BOW PULSE"[8];   // rising edge
   "IO BITS"."BOW PULSE"[8] := #_w46;
   IF #_w47 THEN "TRIGGER" := TRUE; END_IF;
   #_w48 := #_w1 AND ("IEC_Counter_0_DB".CV = 39);
   IF #_w48 THEN "REVAMP".L30 := "SET VALUE"."PRINT INTERVAL"; END_IF;
   #_w49 := #_w48 AND NOT "IO BITS"."BOW PULSE"[9];   // rising edge
   "IO BITS"."BOW PULSE"[9] := #_w48;
   IF #_w49 THEN "TRIGGER" := TRUE; END_IF;
   IF (((50 <= "BUFF".PROCESS) AND ("BUFF".PROCESS <= 69)) OR ((275 <= "BUFF".PROCESS) AND ("BUFF".PROCESS <= 280))) AND ("IEC_Counter_0_DB".CV = 40) THEN
       "IEC_Counter_0_DB".CV := 40;
   END_IF;
END_REGION

